# B&R Automation Studio project MotionTestBenchMaster (part 4)

```iecst
(*HRM Type*)

TYPE
	HrmFlr_Type : 	STRUCT
		STS_StatusBits : InStatusBitHrm_Type; (*0*)
		STS_1 : UINT; (*2*)
		STS_2 : UINT; (*4*)
		STS_WDCount : UINT; (*6*)
		CConfig_NR_Heads : UINT; (*8*)
		CConfig_MotorDirection : UINT; (*10*)
		CConfig_GearIn : UDINT; (*12*)
		CConfig_GearOut : UDINT; (*16*)
		CConfig_Res_1 : UINT; (*20*)
		CConfig_Res_2 : UINT; (*22*)
		CConfig_Res_3 : UINT; (*24*)
		CSetup_Mode : UINT; (*26*)
		CSetup_Acc : UINT; (*28*)
		CSetup_Dec : UINT; (*30*)
		CSetup_EDec : UINT; (*32*)
		CSetup_Gearing : UINT; (*34*)
		CSetup_JogSpeed : UINT; (*36*)
		CSetup_JogAcc : UINT; (*38*)
		CSetup_JogDec : UINT; (*40*)
		CSetup_Rpm_at_00K : UINT; (*42*)
		CSetup_Rpm_at_05K : UINT; (*44*)
		CSetup_Rpm_at_10K : UINT; (*46*)
		CSetup_Rpm_at_15K : UINT; (*48*)
		CSetup_Rpm_at_20K : UINT; (*50*)
		CSetup_Rpm_at_25K : UINT; (*52*)
		CSetup_Rpm_at_30K : UINT; (*54*)
		CSetup_Rpm_at_35K : UINT; (*56*)
		CSetup_Rpm_at_40K : UINT; (*58*)
		CSetup_Rpm_at_45K : UINT; (*60*)
		CSetup_Rpm_at_50K : UINT; (*62*)
		CSetup_Rpm_at_55K : UINT; (*64*)
		CSetup_Rpm_at_60K : UINT; (*66*)
		CSetup_Rpm_at_65K : UINT; (*68*)
		CSetup_Rpm_at_70K : UINT; (*70*)
		CSetup_Rpm_at_75K : UINT; (*72*)
		CSetup_Rpm_at_80K : UINT; (*74*)
		CSetup_Rpm_at_85K : UINT; (*76*)
		CSetup_Rpm_at_90K : UINT; (*78*)
		CSetup_Rpm_at_95K : UINT; (*80*)
		CSetup_Rpm_at_100K : UINT; (*82*)
		CSetup_Res_1 : UINT; (*84*)
		CSetup_Res_2 : UINT; (*86*)
		CSetup_Res_3 : UINT; (*88*)
		STS_DiagCode : UINT;
		STS_3 : UINT; (*90*)
		STS_4 : UINT; (*92*)
		STS_ProdSpeedRPM : UINT; (*94*)
		STS_ProdSpeedBPH : UINT; (*96*)
		STS_HeadSpeedRPM : UINT; (*98*)
		STS_5 : UINT; (*100*)
		STS_ActualCurrent : DINT; (*102 v1.7.4*)
		Spare_0 : UINT; (*104*)
		Spare_1 : UINT; (*108*)
		Spare_2 : UINT; (*110*)
		Spare_3 : UINT; (*112*)
		Spare_4 : UINT; (*114*)
		Spare_5 : UINT; (*118*)
		Spare_6 : UINT; (*120*)
		Spare_7 : UINT; (*122*)
		Spare_8 : UINT; (*124*)
		Spare_9 : UINT; (*126*)
	END_STRUCT;
	FlrHrm_Type : 	STRUCT
		CMD_CommandBits : OutCMDHrm_Type; (*0*)
		CMD_1 : UINT; (*2*)
		CMD_2 : UINT; (*4*)
		CMD_3 : UINT; (*6*)
		CConfig_NR_Heads : UINT; (*8*)
		CConfig_MotorDirection : UINT; (*10*)
		CConfig_GearIn : UDINT; (*12*)
		CConfig_GearOut : UDINT; (*16*)
		CConfig_Res_1 : UINT; (*20*)
		CConfig_Res_2 : UINT; (*22*)
		CConfig_Res_3 : UINT; (*24*)
		CSetup_Mode : UINT; (*26*)
		CSetup_Acc : UINT; (*28*)
		CSetup_Dec : UINT; (*30*)
		CSetup_EDec : UINT; (*32*)
		CSetup_Gearing : UINT; (*34*)
		CSetup_JogSpeed : UINT; (*36*)
		CSetup_JogAcc : UINT; (*38*)
		CSetup_JogDec : UINT; (*40*)
		CSetup_Rpm_at_00K : UINT; (*42*)
		CSetup_Rpm_at_05K : UINT; (*44*)
		CSetup_Rpm_at_10K : UINT; (*46*)
		CSetup_Rpm_at_15K : UINT; (*48*)
		CSetup_Rpm_at_20K : UINT; (*50*)
		CSetup_Rpm_at_25K : UINT; (*52*)
		CSetup_Rpm_at_30K : UINT; (*54*)
		CSetup_Rpm_at_35K : UINT; (*56*)
		CSetup_Rpm_at_40K : UINT; (*58*)
		CSetup_Rpm_at_45K : UINT; (*60*)
		CSetup_Rpm_at_50K : UINT; (*62*)
		CSetup_Rpm_at_55K : UINT; (*64*)
		CSetup_Rpm_at_60K : UINT; (*66*)
		CSetup_Rpm_at_65K : UINT; (*68*)
		CSetup_Rpm_at_70K : UINT; (*70*)
		CSetup_Rpm_at_75K : UINT; (*72*)
		CSetup_Rpm_at_80K : UINT; (*74*)
		CSetup_Rpm_at_85K : UINT; (*76*)
		CSetup_Rpm_at_90K : UINT; (*78*)
		CSetup_Rpm_at_95K : UINT; (*80*)
		CSetup_Rpm_at_100K : UINT; (*82*)
		CSetup_Res_1 : UINT; (*84*)
		CSetup_Res_2 : UINT; (*86*)
		CSetup_Res_3 : UINT; (*88*)
		Spare_0 : UINT; (*90*)
		Spare_1 : UINT; (*92*)
		Spare_2 : UINT; (*94*)
		Spare_3 : UINT; (*96*)
		Spare_4 : UINT; (*98*)
		Spare_5 : UINT; (*100*)
		Spare_6 : UINT; (*102*)
		Spare_7 : UINT; (*104*)
		Spare_8 : UINT; (*106*)
		Spare_9 : UINT; (*108*)
		Spare_10 : UINT; (*110*)
		Spare_11 : UINT; (*112*)
		Spare_12 : UINT; (*114*)
		Spare_13 : UINT; (*116*)
		Spare_14 : UINT; (*118*)
		Spare_15 : UINT; (*120*)
		Spare_16 : UINT; (*122*)
		Spare_17 : UINT; (*124*)
		Spare_18 : UINT; (*126*)
	END_STRUCT;
	InStatusBitHrm_Type : 	STRUCT
		ModeAuto : BOOL; (*From AROL HRM Status Bit - Closure Start command request active*)
		Spare0_1 : BOOL; (*From AROL HRM Status Bit -*)
		Enabled : BOOL; (*From AROL HRM Status Bit - Enable command request active*)
		Spare0_3 : BOOL; (*From AROL HRM Status Bit -*)
		GetDiag_DONE : BOOL; (*From AROL HRM Status Bit - System Diagnostic request executed*)
		Spare0_5 : BOOL; (*From AROL HRM Status Bit -*)
		Ready : BOOL; (*From AROL HRM Status Bit - 1: System Active*)
		Alarm : BOOL; (*From AROL HRM Status Bit -PacDrive Controller Alarm*)
		WatchDog : BOOL; (*From AROL HRM Status Bit -WatchDog signal (1s ON and  1s OFF)*)
		HRM_WR : BOOL; (*From AROL HRM Status Bit -HRM is Writing*)
		ConfigNotOK : BOOL; (*From AROL HRM Status Bit -Configuration is not stored in CompactFlash*)
		SetupNotOK : BOOL; (*From AROL HRM Status Bit -Setup is not stored in CompactFlash*)
		Spare1_4 : BOOL; (*From AROL HRM Status Bit -*)
		Spare1_5 : BOOL; (*From AROL HRM Status Bit -*)
		JogForward : BOOL; (*From AROL HRM Status Bit - Manual Command Forward*)
		JogBackward : BOOL; (*From AROL HRM Status Bit - Manual Command Backward*)
	END_STRUCT;
	OutCMDHrm_Type : 	STRUCT
		ClosureStart : BOOL; (*From AROL HRM Status Bit - Closure Start command request active*)
		Spare0_1 : BOOL; (*From AROL HRM Status Bit -*)
		Enable : BOOL; (*From AROL HRM Status Bit - Enable command request active*)
		Spare0_3 : BOOL; (*From AROL HRM Status Bit -*)
		GetDiag : BOOL; (*From AROL HRM Status Bit - System Diagnostic request executed*)
		Spare0_5 : BOOL; (*From AROL HRM Status Bit -*)
		Reset : BOOL; (*From AROL HRM Status Bit - 1: System Active*)
		Spare0_7 : BOOL; (*From AROL HRM Status Bit -PacDrive Controller Alarm*)
		WatchDog : BOOL; (*From AROL HRM Status Bit -WatchDog signal (1s ON and  1s OFF)*)
		StoreConfig : BOOL; (*From AROL HRM Status Bit -HRM is Writing*)
		StoreSetup : BOOL; (*From AROL HRM Status Bit -Configuration is not stored in CompactFlash*)
		Spare1_3 : BOOL; (*From AROL HRM Status Bit -Setup is not stored in CompactFlash*)
		Spare1_4 : BOOL; (*From AROL HRM Status Bit -*)
		Spare1_5 : BOOL; (*From AROL HRM Status Bit -*)
		JogForward : BOOL; (*From AROL HRM Status Bit - Manual Command Forward*)
		JogBackward : BOOL; (*From AROL HRM Status Bit - Manual Command Backward*)
	END_STRUCT;
END_TYPE

(*Syko Multibody Type*)

TYPE
	FlrSikoMbd_Type : 	STRUCT
		SikoCmd : ARRAY[0..5]OF MotorSikoCmd_Type;
		iWatchDog : INT; (*Input WatchDog*)
	END_STRUCT;
	MbdSikoFlr_Type : 	STRUCT
		SikoSts : ARRAY[0..5]OF MotorSikoSts_Type;
		iWatchDog : INT; (*Input WatchDog*)
	END_STRUCT;
	MotorSikoCmd_Type : 	STRUCT
		xEnable : BOOL; (*Enable motor*)
		xReset : BOOL; (*Reset error*)
		xStartPos : BOOL; (*Start positioning*)
		xJogForward : BOOL; (*Jog forward*)
		xJogBackward : BOOL; (*Jog backward*)
		xSetZero : BOOL; (*Set zero position*)
		xWriteParam : BOOL; (*Write parameter*)
		xReadParam : BOOL; (*Read parameter*)
		wCmdSpare : INT; (*Spare commands word*)
		xTargetPosition : DINT; (*Target position*)
		wPositionVelocity : INT; (*Position velocity*)
		wJogVelocity : INT; (*Jog velocity*)
		bCurrentLimit : BYTE; (*Current limit*)
		bSenseOfRotation : BYTE; (*Sense of rotation*)
		wSpare : INT; (*Sense of rotation*)
		wSpare1 : INT; (*Sense of rotation*)
		wSpare2 : INT; (*Sense of rotation*)
		wSpare3 : INT; (*Sense of rotation*)
	END_STRUCT;
	MotorSikoSts_Type : 	STRUCT
		xPowerOk : BOOL; (*Motor power supply is OK*)
		xEnabled : BOOL; (*Motor is enabled*)
		xReady : BOOL; (*Motor is ready*)
		xRunning : BOOL; (*Motor is running*)
		xInPosition : BOOL; (*Motor is in target position*)
		xBatteryWarning : BOOL; (*Motor battery warning error*)
		xError : BOOL; (*Motor generic error*)
		xSpare_1 : BOOL; (*Spare bit*)
		xParamRwBusy : BOOL; (*Parameter read/write operation is busy*)
		xParamRwError : BOOL; (*Parameter read/write operation is in error*)
		xParamRwDone : BOOL; (*Parameter read/write operation is done*)
		wSpareFdbks : UINT; (*Motor actual position*)
		diActualPosition : DINT; (*Motor actual position*)
		wPositionVelocity : INT; (*Jog velocity*)
		wJogVelocity : INT; (*Current limit*)
		bCurrentLimit : BYTE; (*Sense of rotation*)
		bSenseOfRotation : BYTE;
		wSpare0 : INT;
		wSpare1 : INT;
		wSpare2 : {REDUND_UNREPLICABLE} INT;
		wSpare3 : INT;
	END_STRUCT;
	Head_Diagnostic_Type : 	STRUCT
		FaultNumber : USINT;
		StatusOfInverter : USINT;
		TorqueFeedbackOnHead : UINT;
	END_STRUCT;
END_TYPE

(*WATER TREATMENT V4.A.A.1.6.12*)

TYPE
	FlrWtt_Type : 	STRUCT  (*V4.A.A.1.6.12*)
		Alive : BOOL; (*Life bit signal*)
		ProductionRunning : BOOL;
		ProductRequest : BOOL;
		ProductionAlarm : BOOL; (*V4.A.A.1.7.0*)
		BOOL4 : BOOL;
		BOOL5 : BOOL;
		BOOL6 : BOOL;
		BOOL7 : BOOL;
		CipMode : BOOL; (*V4.A.A.1.7.0*)
		CipAlarm : BOOL; (*V4.A.A.1.7.0*)
		CipProductRequest : BOOL; (*V4.A.A.1.7.0*)
		ControlRunning : BOOL; (*V4.A.A.1.7.0*)
	END_STRUCT;
	WttFlr_Type : 	STRUCT  (*V4.A.A.1.6.12*)
		Alive : BOOL; (*Life bit signal*)
		ProductionMode : BOOL;
		ProductAvailable : BOOL;
		FilterCleaning : BOOL;
		OzoneLevelOk : BOOL;
		BOOL5 : BOOL;
		BOOL6 : BOOL;
		BOOL7 : BOOL;
		CipMode : BOOL; (*V4.A.A.1.7.0*)
		CipAlarm : BOOL; (*V4.A.A.1.7.0*)
		CipSending : BOOL; (*V4.A.A.1.7.0*)
		CheckSolutionOk : BOOL; (*V4.A.A.1.7.0*)
	END_STRUCT;
END_TYPE

(*DATA ACQUISITION COMMUNICATION //V4.A.A.1.6.14*)

TYPE
	FlrDaq_Type : 	STRUCT
		Alive : BOOL;
		StopBit : BOOL; (*Common - Stop bit*)
		OperatorPresence : BOOL; (*Common - Operator presence*)
		ModeAuto : BOOL; (*Common - Operator presence*)
		ModeJog : BOOL; (*Common - Operator presence*)
		ModeSetting : BOOL; (*Common - Operator presence*)
		MachineStatus : UINT; (*Common - Machine Status*)
		SKU : UINT; (*Common - SKU*)
		RecipeNumber : UINT; (*Common - Recipe name*)
		Format : UINT; (*Common - Format*)
		Reason : UDINT; (*Common - Reason code that stop the production on machine*)
		ProductionSpeed : UDINT; (*Common - Production speed in CPM (Container per minute)*)
		SetSpeed : UDINT; (*Common - Set speed*)
		InfeedCount : UDINT; (*Filler - Count of infeed container on the machine*)
		ContainersBurstCount : UDINT; (*Filler - Number of Burst container count*)
		LowLevelEjectCount : UDINT;
	END_STRUCT;
	DaqFlr_Type : 	STRUCT
		Alive : BOOL;
	END_STRUCT;
END_TYPE

(*CODER V4.A.A.1.7.0*)

TYPE
	FlrCdr_Type : 	STRUCT  (*V4.A.A.1.7.1*)
		ProductionRunning : BOOL;
		BOOL1 : BOOL;
		BOOL2 : BOOL;
		BOOL3 : BOOL;
		BOOL4 : BOOL;
		BOOL5 : BOOL;
		BOOL6 : BOOL;
		BOOL7 : BOOL;
		BOOL8 : BOOL;
		BOOL9 : BOOL;
	END_STRUCT;
	CdrFlr_Type : 	STRUCT  (*V4.A.A.1.7.1*)
		Alive : BOOL;
		Ready : BOOL; (*Ready*)
		BOOL2 : BOOL;
		BOOL3 : BOOL;
		BOOL4 : BOOL;
		BOOL5 : BOOL;
		BOOL6 : BOOL;
		BOOL7 : BOOL;
		BOOL8 : BOOL;
		BOOL9 : BOOL;
	END_STRUCT;
END_TYPE

(*PST TREATMENT v999hema*)

TYPE
	FlrPst_Type : 	STRUCT
		AliveBit : BOOL; (*Life bit signal*)
		CipSolutionRequest : BOOL;
		CipAlarm : BOOL;
		CipSolutionReturn : BOOL;
		CipRecoveryCompleted : BOOL;
		CipConditionOK : BOOL;
		CipFlipEnded : BOOL;
		CipRunning : BOOL;
		CipDrainCompleted : BOOL;
		CipLevelReached : BOOL;
		RinseRequest : BOOL;
		RinseEnded : BOOL;
		CopRunning : BOOL;
		RinseAfterProdRequest : BOOL;
		RinseAfterProdEnd : BOOL;
		CopHotWaterReq : BOOL;
		CopEnded : BOOL;
		ProductionRunning : BOOL;
		ProductRequest : BOOL;
		ProductionEnded : BOOL;
		ReadyForHeating : BOOL;
		DoserInTemperature : BOOL;
		AVJ201Open : BOOL;
		DoserEmpty : BOOL;
		DoserFull : BOOL;
		ProductRecoveryEnd : BOOL;
		DoserTankLevel : INT;
		DoserTankLevelSP : INT;
		SlurryDoserVolume : INT;
	END_STRUCT;
	PstFlr_Type : 	STRUCT
		AliveBit : BOOL; (*Life bit signal*)
		CipRecipeCompleted : BOOL;
		CipAlarm : BOOL;
		CipProductSending : BOOL;
		CipRecoveryRequest : BOOL;
		CipConditionOK : BOOL;
		CipFlipAllowed : BOOL;
		CipRunning : BOOL;
		CipDrainRequest : BOOL;
		CipRecipeAborted : BOOL;
		CipReturnEnabled : BOOL;
		RinseMode : BOOL;
		RinseSending : BOOL;
		RinseAfterProd : BOOL;
		CopHotWaterSending : BOOL;
		WorkingRinseFromCip : BOOL;
		WorkingHotSanitation : BOOL;
		WorkingCaustic : BOOL;
		WorkingAcid : BOOL;
		WorkingDisinfectant : BOOL;
		ProductionMode : BOOL;
		ProductAvailable : BOOL;
		MinTankLevel : BOOL;
		DrainRequest : BOOL;
		EndProductionReq : BOOL;
		ProductRecoveryRequest : BOOL;
		ProductCompleted : BOOL;
		HeatingWithWater : BOOL;
		ProductAvailableLiters : INT;
		ProductTemperatureSP : INT;
	END_STRUCT;
END_TYPE
```

### MAU_Global.typ
```iecst
(*SafetyCheck*)

TYPE
	SafeLogicStatus_Type : 	STRUCT
		FailSafe : BOOL;
		FirmwareAcknowledge : BOOL;
		NoExecution : BOOL;
		RunDebug : BOOL;
		RunSafe : BOOL;
		SafeKeyExchange : BOOL;
		Scan : BOOL;
		ModuleExchange : UINT;
		ModuleMissing : UINT;
	END_STRUCT;
END_TYPE

(*DUMMY CONTAINERS*)

TYPE
	MAU_DumCon_Type : 	STRUCT
		DataOut : MAU_DumCon_DataOut_Type;
	END_STRUCT;
	MAU_DumCon_DataOut_Type : 	STRUCT
		Idle : BOOL;
		InstallDone : BOOL;
		RemoveDone : BOOL;
		FixSpeedRequest : BOOL;
		MachineStart : BOOL;
		MachineStop : BOOL;
		CounterEnable : BOOL;
		FmcCipMode : BOOL;
		InsControl : BOOL;
		DisControl : BOOL;
		InsertionPistonFault : BOOL;
		DmcInsCsrPositioning : BOOL;
		DmcDisCsrPositioning : BOOL;
		LftCenteringCupUp : BOOL;
		LftCenteringCupDownOnCip : BOOL;
		ContainerStop : BOOL; (*//1.63*)
		DmcManualModeActive : BOOL; (*v1.6*)
		FlrToCipHeight : BOOL; (*v999*)
		Sector1DownToCip : BOOL; (*v999*)
		Sector2DownToCip : BOOL; (*v999*)
		Sector1DownToProd : BOOL; (*v999*)
		Sector2DownToProd : BOOL; (*v999*)
		Sector1OnlyRotToCip : BOOL;
		Sector2OnlyRotToCip : BOOL;
		Sector2OnlyRotToProd : BOOL;
		Sector1OnlyRotToProd : BOOL;
		DmcUpInProgress : BOOL;
		FillerReversePosReq : BOOL; (*v999*)
		FillerFirstHalfPosReq : BOOL; (*v999*)
		FirstHalfDisDmcControl : BOOL; (*v999*)
		FillerSecondHalfInserted : BOOL;
		FillerFirstHalfRemoved : BOOL;
		FillerFirstHalfInserted : BOOL;
		FillerSecondHalfRemoved : BOOL;
		SecondHalfDisDmcControl : BOOL; (*v999*)
		FirstHalfInsDmcControl : BOOL; (*V999*)
		ManualAirDischarge : BOOL; (*v999*)
		FmcPhasingReq : BOOL; (*v999*)
		FmcInOperational : BOOL; (*v999*)
		FirstHalfInstControl : BOOL; (*v999*)
		SecondHalfInsDmcControl : BOOL; (*v999*)
		FillerSecondHalfPosReq : BOOL; (*v999*)
		FillerSecondReversePosReq : BOOL; (*v999*)
		SectorDiscargePressure : BOOL; (*v999*)
		ContainerLiftAirDischarge : BOOL;
		ManualModeEnableSec2 : BOOL;
		ManualModeEnableSec1 : BOOL;
		DmcManualOperationEn : BOOL; (*V4.A.A.1.7.1*)
		Dba_Sector2ManDownReq : BOOL;
		Dba_Sector1ManDownReq : BOOL;
		ManModeDisControlSec1 : BOOL;
		CycleFmcInError : BOOL;
		CycleAborted : BOOL;
		ReducePressureToUp : BOOL;
		TankCammaToProdHeight : BOOL;
		ManModeDisControlSec2 : BOOL;
	END_STRUCT;
END_TYPE

(*LIFT CONTAINERS*)

TYPE
	MAU_LftCon_Type : 	STRUCT
		DataOut : MAU_LftCon_DataOut_Type;
	END_STRUCT;
	MAU_LftCon_DataOut_Type : 	STRUCT
		LiftContainerUp : BOOL := TRUE;
		CenteringCupUp : BOOL;
		CenteringCupDownOnCip : BOOL;
		CenteringCupAirOn : BOOL := TRUE;
		CenteringCupUpTime : UINT;
		WaterReq : BOOL;
	END_STRUCT;
END_TYPE

(*TRAY*)

TYPE
	MAU_Tray_Type : 	STRUCT  (*v1.4*)
		DataOut : MAU_Tray_DataOut_Type;
	END_STRUCT;
	MAU_Tray_DataOut_Type : 	STRUCT  (*v1.4*)
		ContainerStop : BOOL; (*//1.63*)
		TrayInPosition : BOOL;
	END_STRUCT;
END_TYPE

(*UPS*)

TYPE
	MAU_Ups_Type : 	STRUCT
		DataOut : MAU_Ups_DataOut_Type;
	END_STRUCT;
	MAU_Ups_DataOut_Type : 	STRUCT
		PowerOffTime : UINT;
	END_STRUCT;
END_TYPE

(*AUX  V1.7.2*)

TYPE
	MAU_Aux_Type : 	STRUCT
		DataOut : MAU_Aux_DataOut_Type;
	END_STRUCT;
	MAU_Aux_DataOut_Type : 	STRUCT
		ContainerStop : BOOL;
		EjectionRequest : BOOL;
	END_STRUCT;
END_TYPE

(*SCHEDULER //v1.7.4*)

TYPE
	MAU_Scheduler_Type : 	STRUCT
		DataOut : MAU_Scheduler_DataOut_Type;
	END_STRUCT;
	MAU_Scheduler_DataOut_Type : 	STRUCT
		AlarmMSInternal : UINT;
		AlarmCSRInternal : UINT;
		AlarmCSAInternal : UINT;
		AlarmMSExternal : UINT;
		AlarmCSRExternal : UINT;
		AlarmCSRExternalDw : UINT;
		AlarmCSAExternal : UINT;
		AlarmCSAExternalDw : UINT;
		AlarmInternalOMAC : UINT; (*V1.7.4*)
		AlarmExternalOMAC : UINT; (*V1.7.4*)
	END_STRUCT;
END_TYPE
```

### MC_Global.typ
```iecst
(*Motion Interface Data Type*)

TYPE
	ST_MotionInterface : 	STRUCT
		Safety : ST_SafetyInterface;
		Network : ST_NetworkInterface;
	END_STRUCT;
END_TYPE

(*Interfaces*)

TYPE
	ST_SafetyInterface : 	STRUCT  (*Process-Motion safety interface*)
		Filler : ST_FillerSafetyInterface; (*Filler input/output safety interface*)
		Inlet : ST_InletSafetyInterface; (*Inlet input/output safety interface*)
		Outlet : ST_OutletSafetyInterface; (*Outlet input/output safety interface*)
	END_STRUCT;
	ST_NetworkInterface : 	STRUCT  (*Process-Motion network interface*)
		Machine : ST_MachineInterface; (*Machine input output interface*)
		Inlet : ST_InletInterface; (*Inlet input/output interface*)
		Filler : ST_FillerInterface; (*Filler input/output interface*)
		Outlet : ST_OutletInterface; (*Outlet input/output interface*)
	END_STRUCT;
END_TYPE

(*Machine*)

TYPE
	ST_MachineInterface : 	STRUCT  (*Machine input/output interface structure*)
		Commands : ST_MachineCommandsInterface; (*Machine commands structure*)
		Parameters : ST_MachineParametersInterface; (*Machine parameter structure*)
		Status : ST_MachineStatusInterface; (*Machine status structure*)
		Exceptions : ST_MachineExceptionsInterface; (*Machine exception structure*)
	END_STRUCT;
	ST_MachineCommandsInterface : 	STRUCT  (*Machine commands*)
		HandShakeIn : BOOL; (*Not Used on Full B&R Machines.*)
		MachineStart : BOOL; (*Start commands. When this signal falls the machine start a deceleration ramp.*)
		AlarmReset : BOOL; (*Reset motion alarm command.*)
		MachineQuickStop : BOOL; (*Machine quick stop. This signal has to be set to 1 during normal operation. If this signal will fall a quick stop is performed.*)
		SynchroDisengage : BOOL; (*The interfaces between filler machine and other machines. This value is taken in account only if the CFG_MC.Generic.DisengageImmediately is set.*)
		JogPushButton : BOOL; (*Jog Push Button.*)
		DisableRinserAxis : BOOL; (*The selected axis is disabled rotation V4.A.A.1.7.0*)
		DisableSelectedAxis : BOOL; (*The selected axis is disabled. This operation works only in emergency.*)
		BrakeReleaseModalityRequest : BOOL; (*Brake Release modality request on selected axis.*)
		SelectiveHomeModalityRequest : BOOL; (*Home modality request on selected axis / external reference.*)
		AllAxesHomeModalityRequest : BOOL; (*Homing of all axes - Not Implemented yet.*)
		MultiModalityRequest : BOOL; (*Multi modality selected in order to send the command directly to the module.*)
		PositioningModalityRequest : BOOL; (*Positioning Modality Request.*)
		AutoModalityRequest : BOOL; (*Auto (stand alone) Modality Request.*)
		AutoCombiModalityRequest : BOOL; (*Combi modality request. The machine will follow an external reference.*)
		JogMachineModalityRequest : BOOL; (*Jog modality request.*)
		StepByStepSingleAxisRevModReq : BOOL; (*Single Axis Step By Step Reverse modality request V999*)
		StepByStepSingleAxisModReq : BOOL; (*Single Axis Step By Step modality request V4.A.A.1.7.0*)
		StepByStepModalityRequest : BOOL; (*Step By Step modality request.*)
		EndlessModalityRequest : BOOL; (*Endless modality request - not implemented yet.*)
		ThirdPartMotStatSetupModReq : BOOL; (*Third Party Motor Static Modality Request - not implemented yet.*)
		ThirdPartMotDynSetupModReq : BOOL; (*Endless modality request- not implemented yet.*)
		InMotionTimerModReq : BOOL; (*InMotion Timer function request on active axis.*)
		VelocityModalityRequest : BOOL; (*Velocity Modality Request on actis axis.*)
		OkToDisengage : BOOL; (*The interface is free.*)
		CombiSynchroStop : BOOL; (*Combi Synchro Stop. The machine will continue to turn at constant speed.*)
		MasterEncoderPositionValid : BOOL; (*The position of the master encoder is valid. In case of FALSE in combi mode a Quick Stop is performed.*)
		OnePitchShiftCommand : BOOL; (*One Pitch Shift in combi mode for the "One container every two steps" option.*)
		KochModuleReady : BOOL; (*Where present this variable is linked to the Koch module status*)
		FanSeamerFeedback : BOOL;
		FanSeamerOn : BOOL;
		FanSeamerThermalOverload : BOOL;
	END_STRUCT;
	ST_MachineStatusInterface : 	STRUCT  (*Machine status*)
		HandshakeOut : BOOL; (*Not Used on Full B&R Machines.*)
		MachineHomed : BOOL; (*All axis on the machine are homed.*)
		MachineInPosition : BOOL; (*All axis on the machine are in position.*)
		MachineRunning : BOOL; (*At least one axis is running.*)
		MachineSynchro : BOOL; (*The machine is internally synchronized.*)
		MachineStartFbk : BOOL; (*Feedback of the machine start. See timechart for details.*)
		AutoCmdFeedback : BOOL; (*Auto Modality feedback (?)*)
		JogCmdFeedback : BOOL; (*Jog Modality feedback (?)*)
		AxisNoOp : BOOL;
		MachineIE : BOOL; (*Machine Powered.*)
		MachinePowered : BOOL; (*Machine Powered.*)
		ModuleNotInitialized : BOOL; (*Master Module Not Initialized; the master module isn't initialized. PowerOn the module. 1.7.2a*)
		EnableStart : BOOL; (*Enable start . All motion conditions are ready for the rotation.*)
		EnableAuto : BOOL; (*Enable Auto . All motion conditions are verifier in order to enable auto modality.*)
		EnableEndless : BOOL; (*Enable Endless . All condition are verified in order to have the endless modality.*)
		EnableBrakeRelease : BOOL; (*Enable Brake Release . All condition are verified in order to release the brake.*)
		EnablePositioning : BOOL; (*Enable Positioning . All condition are verified in order to make a positioning.*)
		EnableHoming : BOOL; (*Enable Homing . All condition are verified in order to make the homing of an axis.*)
		EnableCombi : BOOL; (*Enable Combi . All condition are verified in order to enable the combi modality.*)
		EnableMulti : BOOL; (*Enable Multi . All condition are verified in order to enable the spliltted modalities.*)
		EnableSlowMotion : BOOL; (*Enable Slow Motion. All condition are verified in order to enable the slow motion.*)
		EnableStepByStep : BOOL; (*Enable StepByStep . All condition are verified in order to enable the step by step modality.*)
		EnableJog : BOOL; (*Enable Jog . All condition are verified in order to enable the jog modality.*)
		EnableInMotionTimer : BOOL; (*Enable InMotion Timer . All condition are verified in order to enable the in motion timer.*)
		EnableAxisEnable : BOOL; (*Enable AxisEnable Button . All condition are verified in order to enable or disable the axis.*)
		EnableVelocity : BOOL; (*Enable Velocity . All condition are verified in order to make a velociy.*)
		ThirdPartMotStatSetupButton : BOOL; (*Enable thirdy party motor setup. All condition are verified in order to enable the third party static motor setup.*)
		ThirdPartMotDynSetupButton : BOOL; (*Enable thirdy party motor setup. All condition are verified in order to enable the third party dinamic motor setup.*)
		InductionMotSetupButton : BOOL; (*Induction motor setup. All condition are verified in order to enable the third party dinamic motor setup.*)
		NoModalityActive : BOOL; (*No modality selected on motion control.*)
		SelectiveHomeModalityActive : BOOL; (*Selective home modality active.*)
		VelocityModalityActive : BOOL; (*Velocity modality active on axis with velocity control.*)
		PositioningModalityActive : BOOL; (*Positioning modality active.*)
		JogModalityActive : BOOL; (*Jog modality active.*)
		BrakeReleaseModalityActive : BOOL; (*Brake release modality active.*)
		StepByStepSingleAxisRevModActive : BOOL; (*Single Axis Step by step Reverse modality active. V999*)
		StepByStepSingleAxisModeActive : BOOL; (*Single Axis Step by step modality active. V4.A.A.1.7.0*)
		StepByStepModalityActive : BOOL; (*Step by step modality active.*)
		EndlessModalityActive : BOOL; (*Endless modality active.*)
		MultiModalityActive : BOOL; (*Multi modality active. All modules are working indipendently.*)
		ThirdPartMotStatSetupModAct : BOOL; (*Third party motor static setup active.*)
		ThirdPartMotDynSetupModAct : BOOL; (*Third party motor dynamic setup active.*)
		InductionMotSetupActive : BOOL; (*Induction motor setup active.*)
		AutoModalityActive : BOOL; (*Auto modality active.*)
		AutoCombiModalityActive : BOOL; (*Auto combi modality active.*)
		CombiSynchroStopDone : BOOL; (*Combi synchro stop done.*)
		CombiSynchronized : BOOL; (*Combi synchron. All axis are syncrhonized with the external reference.*)
		CombiSynchroInProgress : BOOL; (*Combi synchro in progress.*)
		CombiFixedSpeed : BOOL; (*Combi fixed speed. The combi after a request is running in continous motion.*)
		InMotionTimerDone : BOOL; (*The in motion timer movement has beed done.*)
		OnePitchShiftDone : BOOL;
		MachineClockA : BOOL; (*Main machine clock.*)
		MachineClockB : BOOL; (*Main machine clock.*)
		Clock01 : BOOL; (*Clock 1 at disposal.*)
		Clock02 : BOOL; (*Clock 2 at disposal.*)
		Clock03 : BOOL; (*Clock 3 at disposal.*)
		Clock04 : BOOL; (*Clock 4 at disposal.*)
		Clock05 : BOOL; (*Clock 5 at disposal.*)
		Clock06 : BOOL; (*Clock 6 at disposal.*)
		Clock07 : BOOL; (*Clock 7 at disposal.*)
		Clock08 : BOOL; (*Clock 8 at disposal.*)
		Clock09 : BOOL; (*Clock 9 at disposal.*)
		Clock10 : BOOL; (*Clock 10 at disposal.*)
		Clock11 : BOOL; (*Clock 11 at disposal. v999hema*)
		Clock01AdvStep : BOOL; (*Clock 2 at disposal.*)
		Clock02AdvStep : BOOL; (*Clock 2 at disposal.*)
		Clock03AdvStep : BOOL; (*Clock 3 at disposal.*)
		Clock04AdvStep : BOOL; (*Clock 4 at disposal.*)
		Clock05AdvStep : BOOL; (*Clock 5 at disposal.*)
		Clock06AdvStep : BOOL; (*Clock 6 at disposal.*)
		Clock07AdvStep : BOOL; (*Clock 7 at disposal.*)
		Clock08AdvStep : BOOL; (*Clock 8 at disposal.*)
		Clock09AdvStep : BOOL; (*Clock 9 at disposal.*)
		Clock10AdvStep : BOOL; (*Clock 10 at disposal.*)
		Clock11AdvStep : BOOL; (*Clock 11 at disposal. v999hema*)
		AxisSelectedForEndless : INT; (*Axis selected for endlessfeed feedback.*)
		SpeedForAxisSelectedEndless : INT; (*Speed selected for endlessfeed feedback.*)
		ActualSpeed : REAL; (*Machine velocity [bph].*)
		MachineMaxSpeed : REAL; (*Machine Max velocity [bph].*)
		MachinePitch : REAL; (*Machine Pitch [teens of mm].*)
	END_STRUCT;
	ST_MachineParametersInterface : 	STRUCT  (*Machine parameters*)
		AxisSelectedOnHmi : INT; (*Axis Selected On Hmi*)
		StepNumber : INT; (*Number of step for StepByStep movement [n]*)
		ManualVelocity : UINT;
		JogSpeed : REAL; (*Jog velocity [cph]*)
		AutoSpeed : REAL; (*Auto Velocity [cph]*)
		AutoAccelerationTime : REAL; (*Deceleration Time [s]*)
		AutoDecelerationTime : REAL; (*Acceleration Time [s]*)
		OffsetPositioning : REAL; (*Positioning Offset [mm]*)
		OffsetHoming : REAL; (*Homing Offset - not implemented yet*)
		StopPosition : REAL; (*Stop Position [mm]*)
		InMotionTimerValue : REAL; (*In motion timer value [mm]*)
		Cam01OnValue : REAL; (*Cam01 On Value*)
		Cam01OffValue : REAL; (*Cam01 Off Value*)
		Cam01AdvTime : REAL; (*Cam01 Advance Time*)
		Cam01Pulse : USINT; (*Cam01 Pulse number*)
		Cam02OnValue : REAL; (*Cam02 On Value*)
		Cam02OffValue : REAL; (*Cam02 Off Value*)
		Cam02AdvTime : REAL; (*Cam02 Advance Time*)
		Cam02Pulse : USINT; (*Cam02 Pulse number*)
		Cam03OnValue : REAL; (*Cam03 On Value*)
		Cam03OffValue : REAL; (*Cam03 Off Value*)
		Cam03AdvTime : REAL; (*Cam03 Advance Time*)
		Cam03Pulse : USINT; (*Cam03 Pulse number*)
		Cam04OnValue : REAL; (*Cam04 On Value*)
		Cam04OffValue : REAL; (*Cam04 Off Value*)
		Cam04AdvTime : REAL; (*Cam04 Advance Time*)
		Cam04Pulse : USINT; (*Cam04 Pulse number*)
		Cam05OnValue : REAL; (*Cam05 On Value*)
		Cam05OffValue : REAL; (*Cam05 Off Value*)
		Cam05AdvTime : REAL; (*Cam05 Advance Time*)
		Cam05Pulse : USINT; (*Cam05 Pulse number*)
		Cam06OnValue : REAL; (*Cam06 On Value*)
		Cam06OffValue : REAL; (*Cam06 Off Value*)
		Cam06AdvTime : REAL; (*Cam06 Advance Time*)
		Cam06Pulse : USINT; (*Cam06 Pulse number*)
		Cam07OnValue : REAL; (*Cam07 On Value*)
		Cam07OffValue : REAL; (*Cam07 Off Value*)
		Cam07AdvTime : REAL; (*Cam07 Advance Time*)
		Cam07Pulse : USINT; (*Cam07 Pulse number*)
		Cam08OnValue : REAL; (*Cam08 On Value*)
		Cam08OffValue : REAL; (*Cam08 Off Value*)
		Cam08AdvTime : REAL; (*Cam08 Advance Time*)
		Cam08Pulse : USINT; (*Cam08 Pulse number*)
		Cam09OnValue : REAL; (*Cam09 On Value*)
		Cam09OffValue : REAL; (*Cam09 Off Value*)
		Cam09AdvTime : REAL; (*Cam09 Advance Time*)
		Cam09Pulse : USINT; (*Cam09 Pulse number*)
		Cam10OnValue : REAL; (*Cam10 On Value*)
		Cam10OffValue : REAL; (*Cam10 Off Value*)
		Cam10AdvTime : REAL; (*Cam10 Advance Time*)
		Cam10Pulse : USINT; (*Cam10 Pulse number*)
		Cam11OffValue : REAL; (*Cam11 Off Value v999hema*)
		Cam11AdvTime : REAL; (*Cam11 Advance Time*)
		Cam11OnValue : REAL; (*Cam11 On Value*)
		Cam11Pulse : USINT; (*Cam11 Pulse number*)
		AxisSelectedForEndless : INT; (*Axis Selected for EndlessFeed - not implemented yet*)
		SpeedForAxisSelectedEndless : INT; (*Speed For Axis Selected for EndlessFeed - not implemented yet*)
		MachinePitch : REAL; (*Machine Pitch [teens of mm]*)
	END_STRUCT;
	ST_MachineExceptionsInterface : 	STRUCT  (*Machine exceptions*)
		Fault : BOOL; (*Generic motion exception.*)
		TrackErrorDataException : BOOL;
		HmiChecksumException : BOOL; (*Hmi parameter checksum exception. Used in standalone applications.*)
		PowerSupplyLowMachineException : BOOL; (*Power supply voltage too low exception.*)
		DcBusLowMachineException : BOOL; (*DcBus too low exception.*)
		PhaseMonitoringException : BOOL; (*Phase monitoring exception*)
		KochModuleNotReady : BOOL; (*Where is installed the Koch module ins't correctly charged.*)
		FanSeamearFault : BOOL;
		ExcessiveVelocityException : BOOL; (*Excessive velocity exception (not implemented yet).*)
		ExcessiveAccException : BOOL; (*Excessive acceleration exception (not implemented yet).*)
		NoAxisEnabledException : BOOL; (*No axis enable exception (not implemented yet).*)
		HomingException : BOOL; (*Machine not homed exception.*)
		BleederException : BOOL; (*Bleeder exception. A bleeder error has occurred.*)
		NegativeSpeedBlowerException : BOOL; (*The reference has a negative speed.*)
		CombiException : BOOL;
		InitEncoderException : BOOL;
		FaultCamGeneration : BOOL; (*V1.7.2*)
		StopBlowerException : BOOL;
	END_STRUCT;
END_TYPE

(*Inlet module*)

TYPE
	ST_InletInterface : 	STRUCT  (*Inlet module input/output interface structure*)
		Commands : ST_InletCommands; (*Inlet commands structure*)
		Parameters : ST_InletParameters; (*Inlet parameters structure*)
		Status : ST_InletStatus; (*Inlet status structure*)
		Exceptions : ST_InletExceptions; (*Inlet exception structure*)
	END_STRUCT;
	ST_InletCommands : 	STRUCT  (*Inlet module commands*)
		AutoInletModule : BOOL; (*Auto modality request for auto module in multi mode.*)
		JogInletModule : BOOL; (*Jog modality request for auto module in multi mode.*)
		QuickStopInletModule : BOOL; (*Quick stop on Inlet module; quick stop not active signal 1.*)
		StartInletModule : BOOL; (*Start on Inlet module.*)
		JogPushButtonInletModule : BOOL; (*Jog push button for Inlet module.*)
		SlowMotionBackward : BOOL; (*Slow motion backward on Inlet module.*)
		SlowMotionForward : BOOL; (*Slow motion forward on Inlet module.*)
		AbsolutePositionSensor : BOOL;
		VelocityAxisStop : BOOL;
	END_STRUCT;
	ST_InletStatus : 	STRUCT  (*Inlet module parameters*)
		ModuleHomed : BOOL; (*Inlet Module Homed; all axes are homed.*)
		ModuleInPosition : BOOL; (*Inlet Module In Position; all axes are standstill and in position.*)
		ModuleRunning : BOOL; (*Inlet Module Running; at least one axis is not standstill.*)
		ModulePowered : BOOL; (*Inlet Module Powered; Inlet module is enabled from a safety point of view.*)
		EnableAutoModality : BOOL; (*Inlet Module Enable Auto Modality; during machine multi mode all condition are valid for enabling the Auto modality.*)
		EnableJogModality : BOOL; (*Inlet Module Enable Auto Modality; during machine multi mode all condition are valid for enabling the Jog modality.*)
		ModuleJogActive : BOOL; (*Inlet Module Jog Active; the jog modality on the Inlet module is active.*)
		AutoActive : BOOL; (*Inlet Module Auto Active; the auto modality on the Inlet module is active.*)
		SlowMotionActive : BOOL; (*Inlet Module Slow Motion Active; the slow motion on the Inlet module is active.*)
		JogCmdFeedback : BOOL; (*Inlet Module Jog Command Feedback.*)
		AutoCmdFeedback : BOOL; (*Inlet Module Auto Command Feedback.*)
		ModuleNotInitialized : BOOL; (*Inlet Module Not Initialized; the Inlet module isn't initialized. PowerOn the module.*)
		ModuleReal : BOOL; (*Inlet Module Real; at least one axis is real on the Inlet module.*)
		In01Real : BOOL; (*Axis Inlet01 on filler module is real.*)
		In02Real : BOOL; (*Axis Inlet02 on filler module is real.*)
		In03Real : BOOL; (*Axis Inlet03 on filler module is real.*)
		In04Real : BOOL; (*Axis Inlet04 on filler module is real.*)
		In05Real : BOOL; (*Axis Inlet05 on filler module is real.*)
		In06Real : BOOL; (*Axis Inlet06 on filler module is real.*)
		MainAxisReal : BOOL; (*Main axis on filler module is real.*)
		Velocity : REAL; (*Auto speed for Inlet module [bph].*)
		AbsolutePosition : LREAL;
		AbsolutePositionValid : BOOL;
	END_STRUCT;
	ST_InletParameters : 	STRUCT  (*Inlet module exception*)
		AutoSpeedInletModule : REAL; (*Auto speed for inlet module [bph]*)
		AbsolutePositionValveOffset : UINT;
		ConveyorKs : REAL;
		WheelValvesNumber : UINT;
		TorqueError : CFG_InletTorque_Type;
	END_STRUCT;
	ST_InletExceptions : 	STRUCT  (*Inlet module exception*)
		MainAxisTrackException : BOOL; (*Main Axis Inlet module track error exception.*)
		MainAxisHomeException : BOOL; (*Main Axis Inlet module home exception.*)
		MainAxisTorqueException : BOOL; (*Main Axis Inlet module torque exception.*)
		MainAxisDriveException : BOOL; (*Main Axis Inlet module drive exception.*)
		MainAxisTemperatureError : BOOL; (*Main Axis Inlet module temperature exception.*)
		MainAxisSafetyException : BOOL; (*Main Axis Inlet module safety exception.*)
		MainAxisNotInOpException : BOOL; (*Main Axis Inlet module not in operational exception.*)
		Inlet01TrackException : BOOL; (*Inlet01 track error exception.*)
		Inlet01HomeException : BOOL; (*Inlet01 home exception.*)
		Inlet01TorqueException : BOOL; (*Inlet01 torque exception.*)
		Inlet01DriveException : BOOL; (*Inlet01 drive exception.*)
		Inlet01TemperatureError : BOOL; (*Inlet01 temperature exception.*)
		Inlet01SafetyException : BOOL; (*Inlet01 safety exception.*)
		Inlet01NotInOpException : BOOL; (*Inlet01 not in operational exception.*)
		Inlet02TrackException : BOOL; (*Inlet02 track error exception.*)
		Inlet02HomeException : BOOL; (*Inlet02 home exception.*)
		Inlet02TorqueException : BOOL; (*Inlet02 torque exception.*)
		Inlet02DriveException : BOOL; (*Inlet02 drive exception.*)
		Inlet02TemperatureError : BOOL; (*Inlet02 temperature exception.*)
		Inlet02SafetyException : BOOL; (*Inlet02 safety exception.*)
		Inlet02NotInOpException : BOOL; (*Inlet02 not in operational exception.*)
		Inlet03TrackException : BOOL; (*Inlet03 track error exception.*)
		Inlet03HomeException : BOOL; (*Inlet03 home exception.*)
		Inlet03TorqueException : BOOL; (*Inlet03 torque exception.*)
		Inlet03DriveException : BOOL; (*Inlet03 drive exception.*)
		Inlet03TemperatureError : BOOL; (*Inlet03 temperature exception.*)
		Inlet03SafetyException : BOOL; (*Inlet03 safety exception.*)
		Inlet03NotInOpException : BOOL; (*Inlet03 not in operational exception.*)
		Inlet04TrackException : BOOL; (*Inlet04 track error exception.*)
		Inlet04HomeException : BOOL; (*Inlet04 home exception.*)
		Inlet04TorqueException : BOOL; (*Inlet04 torque exception.*)
		Inlet04DriveException : BOOL; (*Inlet04 drive exception.*)
		Inlet04TemperatureError : BOOL; (*Inlet04 temperature exception.*)
		Inlet04SafetyException : BOOL; (*Inlet04 safety exception.*)
		Inlet04NotInOpException : BOOL; (*Inlet04 not in operational exception.*)
		Inlet05TrackException : BOOL; (*Inlet05 track error exception.*)
		Inlet05HomeException : BOOL; (*Inlet05 home exception.*)
		Inlet05TorqueException : BOOL; (*Inlet05 torque exception.*)
		Inlet05DriveException : BOOL; (*Inlet05 drive exception.*)
		Inlet05TemperatureError : BOOL; (*Inlet05 temperature exception.*)
		Inlet05SafetyException : BOOL; (*Inlet05 safety exception.*)
		Inlet05NotInOpException : BOOL; (*Inlet05 not in operational exception.*)
		Inlet06TrackException : BOOL; (*Inlet06 track error exception.*)
		Inlet06HomeException : BOOL; (*Inlet06 home exception.*)
		Inlet06TorqueException : BOOL; (*Inlet06 torque exception.*)
		Inlet06DriveException : BOOL; (*Inlet06 drive exception.*)
		Inlet06TemperatureError : BOOL; (*Inlet06 temperature exception.*)
		Inlet06SafetyException : BOOL; (*Inlet06 safety exception.*)
		Inlet06NotInOpException : BOOL; (*Inlet06 not in operational exception.*)
	END_STRUCT;
END_TYPE

(*Filler module*)

TYPE
	ST_FillerInterface : 	STRUCT  (*Filler module input/output interface structure*)
		Commands : ST_FillerCommands; (*Filler commands structure*)
		Parameters : ST_FillerParameters; (*Filler parameters structure*)
		Status : ST_FillerStatus; (*Filler status structure*)
		Exceptions : ST_FillerExceptions; (*Filler exceptions structure*)
	END_STRUCT;
	ST_FillerCommands : 	STRUCT  (*Filler module commands structure*)
		AutoFillerModule : BOOL; (*Auto modality request for auto module in multi mode.*)
		JogFillerModule : BOOL; (*Jog modality request for auto module in multi mode.*)
		QuickStopFillerModule : BOOL; (*Quick stop on filler module; quick stop not active signal 1.*)
		StartFillerModule : BOOL; (*Start on filler module.*)
		JogPushButtonFillerModule : BOOL; (*Jog push button for filler module.*)
		FillerAbsolutePositionSensor : BOOL;
		MotorDisableIndex : ARRAY[CST_FirstFillerModuleAxis..CST_LastFillerModuleAxis]OF BOOL; (*v999 test*)
		DisableFillerAxis : BOOL; (*v999hema*)
		DisableDoserAxis : BOOL; (*V4.A.A.1.7.0*)
		DisableRinserAxis : BOOL; (*V4.A.A.1.7.0*)
		RinserAbsolutePositionSensor : BOOL;
		CapperAbsolutePositionSensor : BOOL;
		CrownerAbsolutePositionSensor : BOOL;
		DoserAbsolutePositionSensor : BOOL;
		VelocityAxisStop : BOOL;
		StepByStepModalityRequest : BOOL;
	END_STRUCT;
	ST_FillerStatus : 	STRUCT  (*Filler module status structure*)
		ModuleHomed : BOOL; (*Filler Module Homed; all axes are homed.*)
		ModuleInPosition : BOOL; (*Filler Module In Position; all axes are standstill and in position.*)
		ModuleRunning : BOOL; (*Filler Module Running; at least one axis is not standstill.*)
		ModulePowered : BOOL; (*Filler Module Powered; filler module is enabled from a safety point of view.*)
		EnableAutoModality : BOOL; (*Filler Module Enable Auto Modality; during machine multi mode all condition are valid for enabling the Auto modality.*)
		EnableJogModality : BOOL; (*Filler Module Enable Auto Modality; during machine multi mode all condition are valid for enabling the Jog modality.*)
		StepByStepModalityActive : BOOL;
		ModuleJogActive : BOOL; (*Filler Module Jog Active; the jog modality on the filler module is active.*)
		AutoActive : BOOL; (*Filler Module Auto Active; the auto modality on the filler module is active.*)
		SlowMotionActive : BOOL; (*Filler Module Slow Motion Active; the slow motion on the filler module is active.*)
		JogCmdFeedback : BOOL; (*Filler Module Jog Command Feedback.*)
		AutoCmdFeedback : BOOL; (*Filler Module Auto Command Feedback.*)
		ModuleNotInitialized : BOOL; (*Filler Module Not Initialized; the filler module isn't initialized. PowerOn the module.*)
		ModuleReal : BOOL; (*Filler Module Real; at least one axis is real on the filler module.*)
		FillerAbsolutePositionValid : BOOL;
		RinserAbsolutePositionValid : BOOL;
		CapperAbsolutePositionValid : BOOL;
		CrownerAbsolutePositionValid : BOOL;
		DoserAbsolutePositionValid : BOOL;
		AxisDisabledFeedBack : ARRAY[CST_FirstFillerModuleAxis..CST_LastFillerModuleAxis]OF BOOL; (*v999 test*)
		DoserAxisDisabled : BOOL; (*v999hema*)
		FillerAxisDisabled : BOOL; (*v999hema*)
		RinserAxisDisabled : BOOL; (*Rinser axis disable answer V4.A.A.1.7.0*)
		In01Real : BOOL; (*Axis Inlet01 on filler module is real.*)
		In02Real : BOOL; (*Axis Inlet02 on filler module is real.*)
		In03Real : BOOL; (*Axis Inlet03 on filler module is real.*)
		In04Real : BOOL; (*Axis Inlet04 on filler module is real.*)
		In05Real : BOOL; (*Axis Inlet05 on filler module is real.*)
		In06Real : BOOL; (*Axis Inlet06 on filler module is real.*)
		In07Real : BOOL; (*Axis Inlet07 on filler module is real.*)
		In08Real : BOOL; (*Axis Inlet08 on filler module is real.*)
		In09Real : BOOL; (*Axis Inlet09 on filler module is real.*)
		In10Real : BOOL; (*Axis Inlet10 on filler module is real.*)
		CarouselReal : BOOL; (*Axis Carousel on filler module is real.*)
		Out01Real : BOOL; (*Axis Outlet01 on filler module is real.*)
		Out02Real : BOOL; (*Axis Outlet02 on filler module is real.*)
		Out03Real : BOOL; (*Axis Outlet03 on filler module is real.*)
		Out04Real : BOOL; (*Axis Outlet04 on filler module is real.*)
		Out05Real : BOOL; (*Axis Outlet05 on filler module is real.*)
		Out06Real : BOOL; (*Axis Outlet06 on filler module is real.*)
		Velocity : REAL; (*Filler module actual velocity [bph]*)
		FillerAbsolutePosition : LREAL;
		RinserAbsolutePosition : LREAL;
		CapperAbsolutePosition : LREAL;
		CrownerAbsolutePosition : LREAL;
		DoserAbsolutePosition : LREAL;
	END_STRUCT;
	ST_FillerParameters : 	STRUCT  (*Filler module parameters structure*)
		AutoSpeedFillerModule : REAL; (*Auto speed for filler module [bph]*)
		FillerStepsNumber : UINT;
		RinserStepsNumber : UINT;
		CapperStepsNumber : UINT;
		CrownerStepsNumber : UINT;
		DoserStepsNumber : UINT;
		FillerAbsolutePositionOffset : UINT;
		RinserAbsolutePositionOffset : UINT;
		CapperAbsolutePositionOffset : UINT;
		CrownerAbsolutePositionOffset : UINT;
		DoserAbsolutePositionOffset : UINT;
		InletConveyorKs : REAL;
		OutletConveyorKs : REAL;
		StepNumber : INT; (*Number of step for StepByStep movement [n]*)
		TorqueError : CFG_FillerTorque_Type;
	END_STRUCT;
	ST_FillerExceptions : 	STRUCT  (*Filler module exception structure*)
		Inlet01TrackException : BOOL; (*Inlet01 track error exception.*)
		Inlet01HomeException : BOOL; (*Inlet01 home exception.*)
		Inlet01TorqueException : BOOL; (*Inlet01 torque exception.*)
		Inlet01DriveException : BOOL; (*Inlet01 drive exception.*)
		Inlet01TemperatureError : BOOL; (*Inlet01 temperature exception.*)
		Inlet01SafetyException : BOOL; (*Inlet01 safety exception.*)
		Inlet01NotInOpException : BOOL; (*Inlet01 not in operational exception.*)
		Inlet02TrackException : BOOL; (*Inlet02 track error exception.*)
		Inlet02HomeException : BOOL; (*Inlet02 home exception.*)
		Inlet02TorqueException : BOOL; (*Inlet02 torque exception.*)
		Inlet02DriveException : BOOL; (*Inlet02 drive exception.*)
		Inlet02TemperatureError : BOOL; (*Inlet02 temperature exception.*)
		Inlet02SafetyException : BOOL; (*Inlet02 safety exception.*)
		Inlet02NotInOpException : BOOL; (*Inlet02 not in operational exception.*)
		Inlet03TrackException : BOOL; (*Inlet03 track error exception.*)
		Inlet03HomeException : BOOL; (*Inlet03 home exception.*)
		Inlet03TorqueException : BOOL; (*Inlet03 torque exception.*)
		Inlet03DriveException : BOOL; (*Inlet03 drive exception.*)
		Inlet03TemperatureError : BOOL; (*Inlet03 temperature exception.*)
		Inlet03SafetyException : BOOL; (*Inlet03 safety exception.*)
		Inlet03NotInOpException : BOOL; (*Inlet03 not in operational exception.*)
		Inlet04TrackException : BOOL; (*Inlet04 track error exception.*)
		Inlet04HomeException : BOOL; (*Inlet04 home exception.*)
		Inlet04TorqueException : BOOL; (*Inlet04 torque exception.*)
		Inlet04DriveException : BOOL; (*Inlet04 drive exception.*)
		Inlet04TemperatureError : BOOL; (*Inlet04 temperature exception.*)
		Inlet04SafetyException : BOOL; (*Inlet04 safety exception.*)
		Inlet04NotInOpException : BOOL; (*Inlet04 not in operational exception.*)
		Inlet05TrackException : BOOL; (*Inlet05 track error exception.*)
		Inlet05HomeException : BOOL; (*Inlet05 home exception.*)
		Inlet05TorqueException : BOOL; (*Inlet05 torque exception.*)
		Inlet05DriveException : BOOL; (*Inlet05 drive exception.*)
		Inlet05TemperatureError : BOOL; (*Inlet05 temperature exception.*)
		Inlet05SafetyException : BOOL; (*Inlet05 safety exception.*)
		Inlet05NotInOpException : BOOL; (*Inlet05 not in operational exception.*)
		Inlet06TrackException : BOOL; (*Inlet06 track error exception.*)
		Inlet06HomeException : BOOL; (*Inlet06 home exception.*)
		Inlet06TorqueException : BOOL; (*Inlet06 torque exception.*)
		Inlet06DriveException : BOOL; (*Inlet06 drive exception.*)
		Inlet06TemperatureError : BOOL; (*Inlet06 temperature exception.*)
		Inlet06SafetyException : BOOL; (*Inlet06 safety exception.*)
		Inlet06NotInOpException : BOOL; (*Inlet06 not in operational exception.*)
		Inlet07TrackException : BOOL; (*Inlet07 track error exception.*)
		Inlet07HomeException : BOOL; (*Inlet07 home exception.*)
		Inlet07TorqueException : BOOL; (*Inlet07 torque exception.*)
		Inlet07DriveException : BOOL; (*Inlet07 drive exception.*)
		Inlet07TemperatureError : BOOL; (*Inlet07 temperature exception.*)
		Inlet07SafetyException : BOOL; (*Inlet07 safety exception.*)
		Inlet07NotInOpException : BOOL; (*Inlet07 not in operational exception.*)
		Inlet08TrackException : BOOL; (*Inlet08 track error exception.*)
		Inlet08HomeException : BOOL; (*Inlet08 home exception.*)
		Inlet08TorqueException : BOOL; (*Inlet08 torque exception.*)
		Inlet08DriveException : BOOL; (*Inlet08 drive exception.*)
		Inlet08TemperatureError : BOOL; (*Inlet08 temperature exception.*)
		Inlet08SafetyException : BOOL; (*Inlet08 safety exception.*)
		Inlet08NotInOpException : BOOL; (*Inlet08 not in operational exception.*)
		Inlet09TrackException : BOOL; (*Inlet09 track error exception.*)
		Inlet09HomeException : BOOL; (*Inlet09 home exception.*)
		Inlet09TorqueException : BOOL; (*Inlet09 torque exception.*)
		Inlet09DriveException : BOOL; (*Inlet09 drive exception.*)
		Inlet09TemperatureError : BOOL; (*Inlet09 temperature exception.*)
		Inlet09SafetyException : BOOL; (*Inlet09 safety exception.*)
		Inlet09NotInOpException : BOOL; (*Inlet09 not in operational exception.*)
		Inlet10TrackException : BOOL; (*Inlet10 track error exception.*)
		Inlet10HomeException : BOOL; (*Inlet10 home exception.*)
		Inlet10TorqueException : BOOL; (*Inlet10 torque exception.*)
		Inlet10DriveException : BOOL; (*Inlet10 drive exception.*)
		Inlet10TemperatureError : BOOL; (*Inlet10 temperature exception.*)
		Inlet10SafetyException : BOOL; (*Inlet10 safety exception.*)
		Inlet10NotInOpException : BOOL; (*Inlet10 not in operational exception.*)
		CarouselTrackException : BOOL; (*Carousel track error exception.*)
		CarouselHomeException : BOOL; (*Carousel home exception.*)
		CarouselTorqueException : BOOL; (*Carousel torque exception.*)
		CarouselDriveException : BOOL; (*Carousel drive exception.*)
		CarouselTemperatureError : BOOL; (*Carousel temperature exception.*)
		CarouselSafetyException : BOOL; (*Carousel safety exception.*)
		CarouselNotInOpException : BOOL; (*Carousel not in operational exception.*)
		Outlet01TrackException : BOOL; (*Outlet01 track error exception.*)
		Outlet01HomeException : BOOL; (*Outlet01 home exception.*)
		Outlet01TorqueException : BOOL; (*Outlet01 torque exception.*)
		Outlet01DriveException : BOOL; (*Outlet01 drive exception.*)
		Outlet01TemperatureError : BOOL; (*Outlet01 temperature exception.*)
		Outlet01SafetyException : BOOL; (*Outlet01 safety exception.*)
		Outlet01NotInOpException : BOOL; (*Outlet01 not in operational exception.*)
		Outlet02TrackException : BOOL; (*Outlet02 track error exception.*)
		Outlet02HomeException : BOOL; (*Outlet02 home exception.*)
		Outlet02TorqueException : BOOL; (*Outlet02 torque exception.*)
		Outlet02DriveException : BOOL; (*Outlet02 drive exception.*)
		Outlet02TemperatureError : BOOL; (*Outlet02 temperature exception.*)
		Outlet02SafetyException : BOOL; (*Outlet02 safety exception.*)
		Outlet02NotInOpException : BOOL; (*Outlet02 not in operational exception.*)
		Outlet03TrackException : BOOL; (*Outlet03 track error exception.*)
		Outlet03HomeException : BOOL; (*Outlet03 home exception.*)
		Outlet03TorqueException : BOOL; (*Outlet03 torque exception.*)
		Outlet03DriveException : BOOL; (*Outlet03 drive exception.*)
		Outlet03TemperatureError : BOOL; (*Outlet03 temperature exception.*)
		Outlet03SafetyException : BOOL; (*Outlet03 safety exception.*)
		Outlet03NotInOpException : BOOL; (*Outlet03 not in operational exception.*)
		Outlet04TrackException : BOOL; (*Outlet04 track error exception.*)
		Outlet04HomeException : BOOL; (*Outlet04 home exception.*)
		Outlet04TorqueException : BOOL; (*Outlet04 torque exception.*)
		Outlet04DriveException : BOOL; (*Outlet04 drive exception.*)
		Outlet04TemperatureError : BOOL; (*Outlet04 temperature exception.*)
		Outlet04SafetyException : BOOL; (*Outlet04 safety exception.*)
		Outlet04NotInOpException : BOOL; (*Outlet04 not in operational exception.*)
		Outlet05TrackException : BOOL; (*Outlet05 track error exception.*)
		Outlet05HomeException : BOOL; (*Outlet05 home exception.*)
		Outlet05TorqueException : BOOL; (*Outlet05 torque exception.*)
		Outlet05DriveException : BOOL; (*Outlet05 drive exception.*)
		Outlet05TemperatureError : BOOL; (*Outlet05 temperature exception.*)
		Outlet05SafetyException : BOOL; (*Outlet05 safety exception.*)
		Outlet05NotInOpException : BOOL; (*Outlet05 not in operational exception.*)
		Outlet06TrackException : BOOL; (*Outlet06 track error exception.*)
		Outlet06HomeException : BOOL; (*Outlet06 home exception.*)
		Outlet06TorqueException : BOOL; (*Outlet06 torque exception.*)
		Outlet06DriveException : BOOL; (*Outlet06 drive exception.*)
		Outlet06TemperatureError : BOOL; (*Outlet06 temperature exception.*)
		Outlet06SafetyException : BOOL; (*Outlet06 safety exception.*)
		Outlet06NotInOpException : BOOL; (*Outlet06 not in operational exception.*)
	END_STRUCT;
END_TYPE

(*Outlet module*)

TYPE
	ST_OutletInterface : 	STRUCT  (*Outlet module input/output interface structure*)
		Commands : ST_OutletCommands; (*Outlet commands structure*)
		Parameters : ST_OutletParameters; (*Outlet parameters structure*)
		Status : ST_OutletStatus; (*Outlet status structure*)
		Exceptions : ST_OutletExceptions; (*Outlet  exceptions structure*)
	END_STRUCT;
	ST_OutletCommands : 	STRUCT  (*Outlet module commands structure*)
		AutoOutletModule : BOOL; (*Auto modality request for auto module in multi mode.*)
		JogOutletModule : BOOL; (*Jog modality request for auto module in multi mode.*)
		QuickStopOutletModule : BOOL; (*Quick stop on Outlet module; quick stop not active signal 1.*)
		StartOutletModule : BOOL; (*Start on Outlet module.*)
		JogPushButtonOutletModule : BOOL; (*Jog push button for Outlet module.*)
		SlowMotionBackward : BOOL; (*Slow motion backward on Outlet module.*)
		SlowMotionForward : BOOL; (*Slow motion forward on Outlet module.*)
		AbsolutePositionSensor : BOOL;
		VelocityAxisStop : BOOL;
	END_STRUCT;
	ST_OutletStatus : 	STRUCT  (*Outlet module status structure*)
		ModuleHomed : BOOL; (*Outlet Module Homed; all axes are homed.*)
		ModuleInPosition : BOOL; (*Outlet Module In Position; all axes are standstill and in position.*)
		ModuleRunning : BOOL; (*Outlet Module Running; at least one axis is not standstill.*)
		ModulePowered : BOOL; (*Outlet Module Powered; Outlet module is enabled from a safety point of view.*)
		EnableAutoModality : BOOL; (*Outlet Module Enable Auto Modality; during machine multi mode all condition are valid for enabling the Auto modality.*)
		EnableJogModality : BOOL; (*Outlet Module Enable Auto Modality; during machine multi mode all condition are valid for enabling the Jog modality.*)
		ModuleJogActive : BOOL; (*Outlet Module Jog Active; the jog modality on the Outlet module is active.*)
		AutoActive : BOOL; (*Outlet Module Auto Active; the auto modality on the Outlet module is active.*)
		SlowMotionActive : BOOL; (*Outlet Module Slow Motion Active; the slow motion on the Outlet module is active.*)
		JogCmdFeedback : BOOL; (*Outlet Module Jog Command Feedback.*)
		AutoCmdFeedback : BOOL; (*Outlet Module Auto Command Feedback.*)
		ModuleNotInitialized : BOOL; (*Outlet Module Not Initialized; the Outlet module isn't initialized. PowerOn the module.*)
		ModuleReal : BOOL; (*Outlet Module Real; at least one axis is real on the Outlet module.*)
		MainAxisReal : BOOL; (*Main axis on filler module is real.*)
		Out01Real : BOOL; (*Axis Outlet01 on filler module is real.*)
		Out02Real : BOOL; (*Axis Outlet02 on filler module is real.*)
		Out03Real : BOOL; (*Axis Outlet03 on filler module is real.*)
		Out04Real : BOOL; (*Axis Outlet04 on filler module is real.*)
		Out05Real : BOOL; (*Axis Outlet05 on filler module is real.*)
		Out06Real : BOOL; (*Axis Outlet06 on filler module is real.*)
		Velocity : REAL; (*Outlet module actual velocity [bph]*)
		AbsolutePosition : LREAL;
		AbsolutePositionValid : BOOL;
	END_STRUCT;
	ST_OutletParameters : 	STRUCT  (*Outlet module parameters structure*)
		AutoSpeedOutletModule : REAL; (*Auto speed for Outlet module [bph].*)
		AbsolutePositionValveOffset : UINT;
		ConveyorKs : REAL;
		WheelValvesNumber : UINT;
		TorqueError : CFG_FillerTorque_Type;
	END_STRUCT;
	ST_OutletExceptions : 	STRUCT  (*Outlet module exception structure*)
		MainAxisTrackException : BOOL; (*Main Axis Outlet module track error exception.*)
		MainAxisHomeException : BOOL; (*Main Axis Outlet module home exception.*)
		MainAxisTorqueException : BOOL; (*Main Axis Outlet module torque exception.*)
		MainAxisDriveException : BOOL; (*Main Axis Outlet module drive exception.*)
		MainAxisTemperatureError : BOOL; (*Main Axis Outlet module temperature exception.*)
		MainAxisSafetyException : BOOL; (*Main Axis Outlet module safety exception.*)
		MainAxisNotInOpException : BOOL; (*Main Axis Outlet module not in operational exception.*)
		Outlet01TrackException : BOOL; (*Outlet01 track error exception.*)
		Outlet01HomeException : BOOL; (*Outlet01 home exception.*)
		Outlet01TorqueException : BOOL; (*Outlet01 torque exception.*)
		Outlet01DriveException : BOOL; (*Outlet01 drive exception.*)
		Outlet01TemperatureError : BOOL; (*Outlet01 temperature exception.*)
		Outlet01SafetyException : BOOL; (*Outlet01 safety exception.*)
		Outlet01NotInOpException : BOOL; (*Outlet01 not in operational exception.*)
		Outlet02TrackException : BOOL; (*Outlet02 track error exception.*)
		Outlet02HomeException : BOOL; (*Outlet02 home exception.*)
		Outlet02TorqueException : BOOL; (*Outlet02 torque exception.*)
		Outlet02DriveException : BOOL; (*Outlet02 drive exception.*)
		Outlet02TemperatureError : BOOL; (*Outlet02 temperature exception.*)
		Outlet02SafetyException : BOOL; (*Outlet02 safety exception.*)
		Outlet02NotInOpException : BOOL; (*Outlet02 not in operational exception.*)
		Outlet03TrackException : BOOL; (*Outlet03 track error exception.*)
		Outlet03HomeException : BOOL; (*Outlet03 home exception.*)
		Outlet03TorqueException : BOOL; (*Outlet03 torque exception.*)
		Outlet03DriveException : BOOL; (*Outlet03 drive exception.*)
		Outlet03TemperatureError : BOOL; (*Outlet03 temperature exception.*)
		Outlet03SafetyException : BOOL; (*Outlet03 safety exception.*)
		Outlet03NotInOpException : BOOL; (*Outlet03 not in operational exception.*)
		Outlet04TrackException : BOOL; (*Outlet04 track error exception.*)
		Outlet04HomeException : BOOL; (*Outlet04 home exception.*)
		Outlet04TorqueException : BOOL; (*Outlet04 torque exception.*)
		Outlet04DriveException : BOOL; (*Outlet04 drive exception.*)
		Outlet04TemperatureError : BOOL; (*Outlet04 temperature exception.*)
		Outlet04SafetyException : BOOL; (*Outlet04 safety exception.*)
		Outlet04NotInOpException : BOOL; (*Outlet04 not in operational exception.*)
		Outlet05TrackException : BOOL; (*Outlet05 track error exception.*)
		Outlet05HomeException : BOOL; (*Outlet05 home exception.*)
		Outlet05TorqueException : BOOL; (*Outlet05 torque exception.*)
		Outlet05DriveException : BOOL; (*Outlet05 drive exception.*)
		Outlet05TemperatureError : BOOL; (*Outlet05 temperature exception.*)
		Outlet05SafetyException : BOOL; (*Outlet05 safety exception.*)
		Outlet05NotInOpException : BOOL; (*Outlet05 not in operational exception.*)
		Outlet06TrackException : BOOL; (*Outlet06 track error exception.*)
		Outlet06HomeException : BOOL; (*Outlet06 home exception.*)
		Outlet06TorqueException : BOOL; (*Outlet06 torque exception.*)
		Outlet06DriveException : BOOL; (*Outlet06 drive exception.*)
		Outlet06TemperatureError : BOOL; (*Outlet06 temperature exception.*)
		Outlet06SafetyException : BOOL; (*Outlet06 safety exception.*)
		Outlet06NotInOpException : BOOL; (*Outlet06 not in operational exception.*)
	END_STRUCT;
END_TYPE

(*Filler Module Safety Interface*)

TYPE
	ST_FillerSafetyInterface : 	STRUCT  (*Filler module input/output safety interface structure*)
		Commands : ST_FillerSafetyCommands; (*Filler safety commands*)
		Status : ST_FillerSafetyStatus; (*Filler safety status*)
	END_STRUCT;
	ST_FillerSafetyCommands : 	STRUCT  (*Filler safety commands*)
		EnableModule : BOOL; (*Hardware enable of Filler Module*)
		AxesDiag : ARRAY[0..CST_LastFillerModuleAxis]OF ST_AxesDiag; (*Diagnostic datapoints for filler module axes*)
	END_STRUCT;
	ST_FillerSafetyStatus : 	STRUCT  (*Filler safety status*)
		ModulePowered : BOOL; (*Filler Module Powered*)
	END_STRUCT;
END_TYPE

(*Inlet Module Safety Interface*)

TYPE
	ST_InletSafetyInterface : 	STRUCT  (*Inlet module input/output safety interface structure*)
		Commands : ST_InletSafetyCommands; (*Inlet safety commands*)
		Status : ST_InletSafetyStatus; (*Inlet safety status*)
	END_STRUCT;
	ST_InletSafetyCommands : 	STRUCT  (*Inlet safety commands*)
		EnableModule : BOOL; (*Hardware enable of inlet module*)
		AxesDiag : ARRAY[0..CST_LastInletModuleAxis]OF ST_AxesDiag; (*Diagnostic datapoints for filler module axes*)
	END_STRUCT;
	ST_InletSafetyStatus : 	STRUCT  (*Inlet safety status
*)
		ModulePowered : BOOL; (*Inlet Module Powered*)
	END_STRUCT;
END_TYPE

(*Outlet Module Safety Interface*)

TYPE
	ST_OutletSafetyInterface : 	STRUCT  (*Outlet module input/output safety interface structure*)
		Commands : ST_OutletSafetyCommands; (*Outlet safety commands
*)
		Status : ST_OutletSafetyStatus; (*Outlet safety status*)
	END_STRUCT;
	ST_OutletSafetyCommands : 	STRUCT  (*Outlet safety commands
*)
		EnableModule : BOOL; (*Hardware enable of outlet module*)
		AxesDiag : ARRAY[0..CST_LastOutletModuleAxis]OF ST_AxesDiag; (*Diagnostic datapoints for filler module axes*)
	END_STRUCT;
	ST_OutletSafetyStatus : 	STRUCT  (*Outlet safety status*)
		ModulePowered : BOOL; (*Outlet Module Powered*)
	END_STRUCT;
END_TYPE

(*Axes Diag Safety Struct*)

TYPE
	ST_AxesDiag : 	STRUCT  (*Structure to be connected directly to Hardware*)
		DI_SafeModuleOK : BOOL; (*Safe Module OK Digital input*)
		DI_STOActive : BOOL; (*Safe Torque Off functionality is active*)
		DI_STO1Active : BOOL; (*Safe Torque Off 1 Active*)
		DI_SOSActive : BOOL; (*Safe Operating Stop is active*)
		DI_SS1Active : BOOL; (*Safe Stop 1 is active*)
		DI_SS2Active : BOOL; (*Safe Stop 2 is active*)
		DI_SLS1Active : BOOL; (*Safe Limited speed 1*)
		DI_Operational : BOOL; (*Drive in operational state*)
		DI_NotErrENC : BOOL; (*Encoder not in error state*)
		DI_NotErrFUNC : BOOL; (*Drive not in functional error*)
	END_STRUCT;
END_TYPE

(*MOTION*)

TYPE
	MC_Type : 	STRUCT
		DataOut : MC_DataOut_Type;
	END_STRUCT;
	MC_DataOut_Type : 	STRUCT
		MachineRunning : BOOL;
		ActualSpeed : REAL;
		MaxSpeed : REAL;
	END_STRUCT;
END_TYPE
```

### MNM_Global.typ
```iecst
(*MAIN DRIVE CONTROL*)

TYPE
	MNM_Type : 	STRUCT
		DataOut : MNM_DataOut_Type;
	END_STRUCT;
	MNM_DataOut_Type : 	STRUCT
		HornFlrRequest : BOOL;
		StartLightBlinkRequest : BOOL;
		StartLightFixRequest : BOOL;
		CopSpeedReqReached : BOOL;
		RnsSpeedReqReached : BOOL;
		CapSpeedReqReached : BOOL;
		DmcSpeedReqReached : BOOL;
		SftSpeedReqReached : BOOL;
		SkidSpeedReqReached : BOOL;
		EmptySpeedReached : BOOL;
		ContBlockSpeedReached : BOOL;
		ContBlock1Requested : BOOL;
		ContBlock2Requested : BOOL;
		MachineRunning : BOOL; (*Module Running*)
		ReadyForVortexCalib : BOOL;
		ReadyForCoupling : BOOL;
		PartnerReadyToRun : BOOL;
		OperatorPresence : BOOL;
		FixSpeedRequest : BOOL;
		OutletSpeed : REAL;
		LackInlet1 : BOOL;
		LackInlet2 : BOOL;
		COPInletContBlockSpeedReached : BOOL;
		ContainerStop : BOOL;
		DesyncroRequest : BOOL;
		CapperPositioningDone : BOOL;
		SingleAxisInPosition : BOOL;
		RinserAxisDisabled : BOOL;
		DoserAxisDisabled : BOOL;
		FillerAxisDisabled : BOOL;
		FillingValvePositioningDone : BOOL;
		ReversePositioningDone : BOOL;
		DmcPositioningDone : BOOL;
		PhaseDone : BOOL;
		ConfigReqLoaded : BOOL;
		StartRequest : BOOL;
		InletSpeed : REAL;
	END_STRUCT;
END_TYPE
```

### MNT_Global.typ
```iecst
(*MAINTENANCE*)

TYPE
	MNT_Type : 	STRUCT  (*v1.4*)
		DataOut : MNT_DataOut_Type;
	END_STRUCT;
	MNT_DataOut_Type : 	STRUCT  (*v1.4*)
		LotoInExecution : BOOL;
		LotoValvesOpening : BOOL;
		LotoAirDischarge : BOOL;
		LotoAirDischargePilot : BOOL;
		LotoDmcOn : BOOL;
		LotoStep : USINT;
		LotoDevices : INT;
	END_STRUCT;
END_TYPE
```

### OPS_Global.typ
```iecst
(*SAFETY*)

TYPE
	OPS_Type : 	STRUCT
		DataOut : OPS_DataOut_Type; (*SAFE_PLC Inputs*)
	END_STRUCT;
	OPS_DataOut_Type : 	STRUCT
		EmergencyOk : BOOL := TRUE;
		FlrDoorsOk : BOOL := TRUE;
		DoorsOk : BOOL;
		GeneralAirOn : BOOL;
		ConfinementZoneRed : BOOL;
		BeaconHornJog : BOOL; (*Blow horn request for jog*)
		FlrModeSelectorAuto : BOOL := TRUE;
		FlrModeSelectorAdjustment : BOOL := TRUE;
		FlrModeSelectorJog : BOOL := TRUE;
		JogStartPb : BOOL := TRUE;
		SelModeChange : BOOL; (*Mode selection Error*)
		EnableDrive : BOOL;
		EnablePump : BOOL;
		EnableProcessValves : BOOL;
		EnableCopValves : BOOL; (*V4.A.A.1.6.11a*)
		EnableVerticalDrive : BOOL; (*V4.A.A.1.6.6*)
		BufferDoorOpened : BOOL;
		BufferDoorFault : BOOL;
		HMIDoorUnlock : BOOL;
		LabellerTrasferDoorOpenRequest : BOOL;
		BlowerTrasferDoorOpenRequest : BOOL;
		ActisTrasferDoorOpenRequest : BOOL; (*V4.A.A.1.6.12*)
		LabellerTrasferGateOpened : BOOL;
		BlowerTrasferGateOpened : BOOL;
		ActisTrasferGateOpened : BOOL; (*V4.A.A.1.6.12*)
		AutomaticInletGate : BOOL; (*Not Used in Glass Machine*)
		InletGateOpened : BOOL; (*V4.A.A.1.6.12h*)
		InletGateClosed : BOOL;
		OutletGateClosed : BOOL;
		OutletGateOpened : BOOL; (*V4.A.A.1.7.0*)
		OperatorPresence : BOOL;
		ContainerStop : BOOL; (*//1.63*)
		ConfigSaveReq : BOOL;
		FlrLiftingEnabled : BOOL;
		FillerLiftPw : BOOL; (*maste nuovo*)
		FillerLiftPwFault : BOOL; (*master nuovo*)
		DoorsOpenExceptGloves : BOOL; (*V4.A.A.1.7.0*)
	END_STRUCT;
END_TYPE
```

### REL_Global.typ
```iecst
(*ELECTRONIC FUSES*)

TYPE
	REL_Type : 	STRUCT
		DataOut : REL_DataOut_Type;
	END_STRUCT;
	REL_DataOut_Type : 	STRUCT
		ElectronicFusesPresence : BOOL;
		GlobalPowerOn : BOOL := TRUE;
		Station : ARRAY[1..16]OF REL_Channel_Type;
	END_STRUCT;
	REL_Channel_Type : 	STRUCT
		Ch : ARRAY[1..16]OF REL_Status_Type;
	END_STRUCT;
	REL_Status_Type : 	STRUCT
		ConfigurationError : BOOL;
		PoweredOn : BOOL;
		Overload : BOOL;
		ShortCircuit : BOOL;
	END_STRUCT;
END_TYPE
```

### RCP_Global.typ
```iecst
(*PRODUCTION RECIPE MANAGER*)

TYPE
	RCP_Type : 	STRUCT
		DataOut : RCP_DataOut_Type;
	END_STRUCT;
	RCP_DataOut_Type : 	STRUCT
		RecipeDownload : BOOL;
		RecipeDownloaded : BOOL;
	END_STRUCT;
END_TYPE
```

### SFT_Global.typ
```iecst
(*CONTAINERS SHIFT REGISTER*)

TYPE
	SFT_Type : 	STRUCT
		DataOut : SFT_DataOut_Type;
	END_STRUCT;
	SFT_DataOut_Type : 	STRUCT
		Alarm : SFT_Alarm_Type;
		ContainersBlock1 : BOOL; (*Block container in corrispondence of FV disable*)
		ContainersBlock2 : BOOL; (*Block container in corrispondence of FV disable*)
		ContainerStop : BOOL; (*//1.63*)
		ContainersReleaseEarlier1 : BOOL;
		ContainersReleaseEarlier2 : BOOL;
		ContainersAtCarouselOutlet : BOOL;
		ContainerAtMachineOutlet : BOOL;
		CombiEmpty : BOOL; (*No containers in the combi*)
		MachineEmpty : BOOL; (*No containers in the machine*)
		_20Bottles_AtExit : BOOL; (*Signals For Conveyor - Information 20 bottles at machine exit*)
		RinserTreatmentRequest : BOOL;
		BottleCoolingRequest : BOOL;
		InletConveyorEmpty : BOOL;
		OutletConveyorEmpty : BOOL;
		CapsAirRequest : BOOL; (*Closing Unit - Air Blow*)
		CapsReleaseProductionReady : BOOL;
		CapsReleaseEmptyingReady : BOOL;
		CapsReleaseEmpty : BOOL; (*v1.5*)
		CappingHeadAtMachineGetData : BOOL; (*V4.A.A.1.6.12*)
		CapOnCappingHead : BOOL; (*v1.5*)
		FMC_PreClosingContainerReq : BOOL;
		FMC_ContainerPresenceReq : BOOL;
		FMC_WashCenteringCup : BOOL;
		FMC_StartFillingReq : BOOL;
		FillingValveRinseReq : BOOL;
		ManPreformLoadingReq : BOOL;
		VBS_Presence : BOOL;
		DmcNotInserted : BOOL;
		DmcNotRemoved : BOOL;
		CounterDone : BOOL;
		ValveDisabledPreformBlock : BOOL;
		ValveDisabledLbrBottleEjection : BOOL;
		SlowDownContBlockReq : BOOL;
		ContBlockSpeedReq : BOOL;
		ManualContainersReleaseEnable : BOOL; (*Block container in corrispondence of FV disable*)
		OutletShowerReq : BOOL;
		NeckRinseReq : BOOL;
		MachineInletStatus : BOOL;
		COPInletContSlowSpeedReq : BOOL;
		COPInletContConvEmptyRunning : BOOL;
		COPInletContConvEmptyDone : BOOL;
		FillingValvePositionReq : BOOL; (*Filling valve positioning request*)
		PreformManualLoading : BOOL; (*v1.6*)
		CapTreatmentStart : BOOL; (*V4.A.A.1.7.0*)
		NoBottleNoSprayPistonFault : BOOL; (*vrma*)
		NoBottleNoSprayActive : BOOL; (*vrma*)
		FirstHalfDmcInsered : BOOL;
		SecondHalfCounterDone : BOOL;
		SecondHalfDmcNotInserted : BOOL;
		SecondHalfDmcNotRemoved : BOOL;
		FillingValveAtMachineInlet : INT;
		CappingHeadAtMachineInlet : INT;
		CapHeadNumberInTangency : INT; (*V4.A.A.1.6.12*)
		RinsingNozzleAtMachineInlet : INT; (*V4.A.A.1.6.12*)
		RinserBypassedPointer : INT; (*V4.A.A.1.6.12*)
		BottleBurstWashRampActivation : ARRAY[1..3]OF BOOL; (*master nuovo*)
		FoamerRequest : BOOL;
		CrownsReleaseProductionReady : BOOL;
		CrownsAirRequest : BOOL;
		FillingValve1 : BOOL; (*FCI:TEST v1.7.4a*)
		CapperHead1 : BOOL; (*FCI:TEST v1.7.4a*)
		CrownerHead1 : BOOL; (*FCI:TEST v1.7.4a*)
		DoserHead1 : BOOL; (*v999hema*)
		AuxBlowerMold1 : BOOL; (*FCI:TEST v1.7.4a*)
		AuxLabelerPlate1 : BOOL; (*FCI:TEST v1.7.4a*)
		ContainersInFiller : UINT; (*Number of containers in the machine*)
		ContainersInConveyorReject : UINT; (*Number of container to be reject after COP vrmaCOP *)
		ContainersInMachine : UINT; (*Number of containers in the machine*)
		ContainersToFillFillerOnly : UINT;
		ContainersToFill : UINT; (*Number of containers to be filled (From Container Block To Inlet Tangency)*)
		ContainersToCap : UINT; (*Number of containers to be filled (From Container Block To Inlet Tangency) V4.A.A.1.7.0*)
		BottleCoolingFillerSteps : UINT;
		RinserFillerSteps : UINT; (*V4.A.A.1.6.12*)
		DoserFillerSteps : UINT; (*v999hema*)
		NumberDmcInserted : UINT;
		FillingValvePosValue : UINT; (*Number of filling valve to position in the ispection point*)
		CopPurgeStep : UINT; (*vrmaCOP*)
		ContBlockSpeedValue : REAL;
		COPInletContBlockSpeedValue : REAL;
		FMC_PreClosingContainerReqByte : USINT; (*v1.7.4*)
		FMC_ContainerPresenceReqByte : USINT; (*v1.7.4*)
		FMC_StartFillingReqByte : USINT; (*v1.7.4*)
		DmcClockSensorBroken : BOOL;
		ChannelEmptyingDone : BOOL; (*vrmaCOP*)
	END_STRUCT;
	SFT_Alarm_Type : 	STRUCT
		BottMissingForFillerFault : BOOL;
		Category : DINT;
		ID : DINT;
		OmacCode : DINT;
	END_STRUCT;
END_TYPE

(*SHIFT*)

TYPE
	MachineShift_Type : 	STRUCT
		ShiftInfo : UINT;
		FillingNozzle : USINT;
		CrownerHead : USINT;
		DoserHead : USINT; (*v999hema*)
		CappingHead : USINT;
		RinsingNozzle : USINT; (*V4.A.A.1.7.0*)
	END_STRUCT;
	CombiShift_Type : 	STRUCT
		MoldNumber : UINT; (*V1.61*)
		CombiInfo : UINT;
		AlarmId : UDINT;
		Category : UDINT;
		OmacCode : UDINT;
	END_STRUCT;
END_TYPE
```

### TNK_Global.typ
```iecst
(*TANK*)

TYPE
	TNK_Type : 	STRUCT
		DataOut : TNK_DataOut_Type;
	END_STRUCT;
	TNK_DataOut_Type : 	STRUCT
		Wait : BOOL;
		CipMode : BOOL;
		CipDrainMode : BOOL;
		RinseMode : BOOL;
		DrainMode : BOOL;
		ProdMode : BOOL;
		PushBackMode : BOOL;
		StartUp : BOOL;
		SipMode : BOOL;
		DeEnergization : BOOL;
		EndProduction : BOOL;
		Calibration : BOOL; (*V4.A.A.1.6.13*)
		ContainerStop : BOOL; (*//1.63*)
		DummyContainersIns : BOOL;
		DummyContainersDis : BOOL;
		CopInProductionActive : BOOL;
		StartUpHOT : BOOL;
		StartCipRinser : BOOL;
		APCORunning : BOOL;
		DisableCipRinser : BOOL;
	END_STRUCT;
END_TYPE
```

### DOS_Global.typ
```iecst
(*FLAVOR DOSER*)

TYPE
	DOS_Type : 	STRUCT
		DataOut : DOS_DataOut_Type;
	END_STRUCT;
	DOS_DataOut_Type : 	STRUCT  (*v999hema*)
		FillingHeatingProd : BOOL;
		FillingProd : BOOL;
		WaitMode : BOOL;
		ProdMode : BOOL;
		ProductRequest : BOOL;
		ProductionEnd : BOOL;
		ReadyForHeating : BOOL;
		DoserFull : BOOL;
		AVJ201Open : BOOL;
		DoserEmpty : BOOL;
		DoserInTemperature : BOOL;
		RecoveryEnd : BOOL;
		EjectionRequest : BOOL;
		HotWaterReq : BOOL;
		NecessaryBottleEndProd : REAL;
		CipMode : BOOL;
		CipConditionOk : BOOL;
		CipSolutionReq : BOOL;
		CipRecovery : BOOL;
		CipRecoveryEnd : BOOL;
		CipAlarm : BOOL;
		RinseEnd : BOOL;
		RinseReq : BOOL;
		CipDrainEnd : BOOL;
		CipLevelReached : BOOL;
		CipSystemFlooded : BOOL;
		RinseAfterProdReq : BOOL;
		RinseMode : BOOL;
		RinseAfterProdEnd : BOOL;
		DrainMode : BOOL;
		CopMode : BOOL;
		CopAfterCipReq : BOOL;
		CopRunning : BOOL;
		AromePodReq : BOOL;
		MachineStart : BOOL;
		MachineStop : BOOL;
		DoserExcluded : BOOL;
		DoserIncluded : BOOL;
		ByPassed : BOOL;
		AxisEnableRequest : BOOL;
		AxisDisableRequest : BOOL;
		FillerAxisDisableRequest : BOOL;
		StepCounterRequest : BOOL;
		FixSpeedRequest : BOOL;
		PositionReached : BOOL;
		CommandToValve : BOOL;
		FixSpeedValue : REAL;
		FillerProdStartEnable : BOOL;
		FillerCipStartEnable : BOOL;
		FillerRinseStartEnable : BOOL;
		PhasingWithDos : BOOL;
		PhasingWithoutDos : BOOL;
	END_STRUCT;
END_TYPE
```

### Sequencer.typ
```iecst
(*SEQUENCER PERMANENT TYPE*)

TYPE
	SEQ_Permanent_Type : 	STRUCT
		SeqActualStep : UINT;
		SeqBackupStep : UINT;
		SeqMode1 : UINT;
		SeqMode2 : UINT;
		SeqAuxiliary : UINT;
	END_STRUCT;
END_TYPE
```

### BTC_Global.typ - not listed in the package file held
```iecst
(*BOTTLE BOTTOM COOLING*)

TYPE
	BTC_Type : 	STRUCT
		DataOut : BTC_DataOut_Type;
	END_STRUCT;
	BTC_DataOut_Type : 	STRUCT
		Idle : BOOL; (*v1.4*)
		StepCountReq : BOOL;
		CipMode : BOOL;
		CipDrainMode : BOOL;
		RinseMode : BOOL;
		DrainMode : BOOL;
		ProdMode : BOOL;
		StartUp : BOOL;
		CopMode : BOOL;
		DeEnergization : BOOL;
		SamplingCommand : BOOL; (*V4.A.A.1.6.12*)
		SamplingInPosition : BOOL; (*V4.A.A.1.6.12*)
		ContainerStop : BOOL; (*//1.63*)
		WaterFlow : REAL;
		Temperature : REAL;
		TemperatureGlicol : REAL; (*V4.A.A.1.7.1*)
	END_STRUCT;
END_TYPE
```

### EIT_Global.typ - not listed in the package file held
```iecst
(*OPC VARIABLES - CHANGE THEM REQUIRES TO CHANGE OPC CONFIGURATION AND A WARM RESTART*)

TYPE
	EIT_Type : 	STRUCT
		Version : INT;
		Reason : DINT; (*Common - Reason code that stop the production on machine*)
		StopBit : BOOL; (*Common - Stop bit*)
		ProductionSpeed : REAL; (*Common - Production speed in CPM (Container per minute)*)
		SetSpeed : REAL; (*Common - Set speed*)
		UnitPerCount : INT; (*Common - Unit Per count*)
		SKU : INT; (*Common - SKU*)
		RecipeName : STRING[80]; (*Common - Recipe name*)
		OperatorPresence : BOOL; (*Common - Operator presence*)
		Format : STRING[20]; (*Common - Format*)
		MachineStatus : USINT; (*Common - Machine Status*)
		Count : EITCount_Type; (*Common - Specific Count tag different for each machine on the EITCount definition*)
		Measure : EITMeasure_Type; (*Common - Specific Measure tag different for each machine on the WITMeasure definition*)
		EZ : EITEZ_Type;
		SBO : EITSBO_Type;
		CapFeed : EITCapFeed_Type; (*Common - Uses for filler with Cap feeder*)
		Capper : EITCapper_Type; (*Common - Uses for filler with capper*)
		RunningEvent : EITRunningEvent_Type;
	END_STRUCT;
	EITCount_NotUsed_Type : 	STRUCT
		FillerRotationTotalizer : DINT; (*Filler - Number of filler revolution*)
		CapperRotationTotalizer : DINT; (*Filler - Number of capper revolution*)
		RinserRotationTotalizer : DINT; (*Filler - Number of rinser revolution*)
		BadFillingCount : DINT; (*Filler - Number of Bad filling count*)
		BadCappingCount : DINT; (*Filler - Number of Bad capping count*)
		BadRinsingCount : DINT; (*Filler - Number of Bad rinsing count*)
		ContainerOut : DINT; (*Filler - Count of container produced*)
		ContainerEjected : DINT; (*Filler - Count of container ejected*)
	END_STRUCT;
	EITCount_Type : 	STRUCT
		InfeedCount : UDINT; (*Filler - Count of infeed container on the machine*)
		ContainersBurstCount : UDINT; (*Filler - Number of Burst container count*)
		ContainersEjectManually : UDINT; (*Filler - Count of container ejected manually*)
		LowLevelEjectCount : UDINT;
		LPCA : UDINT; (*Filler - FlowLPCA V4.A.A.1.6.14k*)
		General_CO2 : UDINT;
		ClosingUnit_CO2 : UDINT;
		N2 : UDINT;
		ProcessWater : UDINT;
		CopWater : UDINT;
		BottleBottomCoolingWater : UDINT; (*V4.A.A.1.6.14k*)
		Product : UDINT;
		Steam : UDINT;
		FoodSteam : UDINT;
		ProductWater : UDINT; (*V4.A.A.1.6.14k*)
		Syrup : UDINT;
		ElectricalEnergy : UDINT; (*V4.A.A.1.6.14k*)
	END_STRUCT;
	EITMeasure_Type : 	STRUCT
		FlowLPCA : REAL; (*Filler - FlowLPCA V4.A.A.1.6.14k*)
		ElectricalPower : REAL; (*Filler - Electrical power KW*)
	END_STRUCT;
	EITEZ_Type : 	STRUCT
		StopBit : BOOL;
		Reason : INT;
	END_STRUCT;
	EITSBO_Type : 	STRUCT
		StopBit : BOOL;
		Reason : INT;
	END_STRUCT;
	EITCapFeed_Type : 	STRUCT
		StopBit : BOOL;
		Reason : INT;
	END_STRUCT;
	EITCapper_Type : 	STRUCT
		StopBit : BOOL;
		Reason : INT;
	END_STRUCT;
	EITRunningEvent_Type : 	STRUCT
		CapsLowLevel : BOOL;
		LidLowLevel : BOOL;
	END_STRUCT;
	EIT_ChangeOver_Type : 	STRUCT
		ToHLI : EIT_ChangeOver_To_Type;
		FromHLI : EIT_ChangeOver_From_Type;
	END_STRUCT;
	EIT_ChangeOver_From_Type : 	STRUCT
		NextProductReady : BOOL;
		PrepareForChange : BOOL;
		RinseRequested : BOOL;
		StopProduction : BOOL;
		WatchDog : INT;
		ProductToLoad : INT;
		NextRecipeId : UDINT;
		RemainingProdToDo : UDINT;
	END_STRUCT;
	EIT_ChangeOver_To_Type : 	STRUCT
		ChangeOverDone : BOOL;
		ChangeOverOptionOn : BOOL;
		ProductionEnded : BOOL;
		NextProductValidationRequest : BOOL;
		WatchDog : INT;
		ActualProduct : INT;
		ActualRecipeId : UDINT;
		ProductionBatchAvailable : UDINT;
	END_STRUCT;
	EIT_OMAC_Type : 	STRUCT
		Status : EIT_PMLs_Type;
		Command : EIT_PMLc_Type;
		Admin : EIT_PLMa_Type;
	END_STRUCT;
	EIT_PLMa_Type : 	STRUCT
		Alarm : EIT_PMLa_Alarm_Type;
	END_STRUCT;
	EIT_PMLa_Alarm_Type : 	STRUCT
		ID : UDINT;
		Value : UDINT;
		Message : STRING[80];
	END_STRUCT;
	EIT_PMLc_Type : 	STRUCT
		New_Member : USINT;
	END_STRUCT;
	EIT_PMLs_Type : 	STRUCT
		UnitModeCurrent : UDINT;
		StateCurrent : UDINT;
	END_STRUCT;
	WS_Type : 	STRUCT
		Communication : WS_Communication_Type;
		Tracking : WS_Tracking_Type;
		OperatingMode : WS_OperatingMode_Type;
		Omac : WS_Omac_Type;
		Fault : WS_Fault_Type;
		Pointer : WS_Pointer_Type;
		Parameter : WS_Parameter_Type;
		Counters : WS_Counters_Type;
	END_STRUCT;
	WS_Communication_Type : 	STRUCT
		WS_Error : UDINT; (*Tag-Number: 00000*)
		WS_PDACONT_Lenght : UDINT; (*Tag-Number: 00001*)
		WS_Test_Unsigned32_1 : UDINT; (*Tag-Number: 00011*)
		WS_Test_Unsigned32_2 : UDINT; (*Tag-Number: 00012*)
		WS_Test_Unsigned32_3 : UDINT; (*Tag-Number: 00013*)
		WS_Test_Signed32_1 : DINT; (*Tag-Number: 00014*)
		WS_Test_Signed32_2 : DINT; (*Tag-Number: 00015*)
		WS_Test_Signed32_3 : DINT; (*Tag-Number: 00016*)
		WS_Test_Real_1 : REAL; (*Tag-Number: 00017*)
		WS_Test_Real_2 : REAL; (*Tag-Number: 00018*)
		WS_Test_Real_3 : REAL; (*Tag-Number: 00019*)
		WS_Test_Hex32_1 : DWORD; (*Tag-Number: 00020*)
		WS_Test_Hex32_2 : DWORD; (*Tag-Number: 00021*)
		WS_Test_Hex32_3 : DWORD; (*Tag-Number: 00022*)
		WS_Test_String16_1 : STRING[1]; (*Tag-Number: 00023*)
		WS_Test_String16_2 : STRING[1]; (*Tag-Number: 00024*)
		WS_Test_String16_3 : STRING[1]; (*Tag-Number: 00025*)
	END_STRUCT;
	WS_Tracking_Type : 	STRUCT
		WS_Set_Batch_ID_L : DINT; (*Tag-Number: 00061*)
		WS_Set_Batch_ID_H : DINT; (*Tag-Number: 00062*)
		WS_Cur_Batch_ID_L : DINT; (*Tag-Number: 00063*)
		WS_Cur_Batch_ID_H : DINT; (*Tag-Number: 00064*)
	END_STRUCT;
	WS_OperatingMode_Type : 	STRUCT
		WS_Cur_Mode : UDINT; (*Tag-Number: 00100*)
		WS_Cur_Prog : UDINT; (*Tag-Number: 00200*)
		WS_Prog_Step : UDINT; (*Tag-Number: 00210*)
		WS_Cur_State : UDINT; (*Tag-Number: 00300*)
	END_STRUCT;
	WS_Omac_Type : 	STRUCT
		WS_Cur_Mach_Spd : REAL; (*Tag-Number: 00401*)
		WS_Set_Mach_Spd : REAL; (*Tag-Number: 00402*)
		WS_Mach_Design_Spd : REAL; (*Tag-Number: 00403*)
		WS_Mach_Cycle : UDINT; (*Tag-Number: 00501*)
		WS_Mat_Ready : DWORD; (*Tag-Number: 00601*)
		WS_Mat_Low : DWORD; (*Tag-Number: 00602*)
		WS_Prod_Ratio : UDINT; (*Tag-Number: 00701*)
	END_STRUCT;
	WS_Fault_Type : 	STRUCT
		WS_Not_Of_Fail_Code : UDINT; (*Tag-Number: 10000*)
	END_STRUCT;
	WS_Pointer_Type : 	STRUCT
		WS_Pointer_Code : UDINT; (*Tag-Number: 20000*)
	END_STRUCT;
	WS_Parameter_Type : 	STRUCT
		WS_Container_Type : UDINT; (*Tag-Number: 30003*)
		WS_Beer_Type : UDINT; (*Tag-Number: 30004*)
	END_STRUCT;
	WS_Measured_Type : 	STRUCT
		WS_Press_Bottling : REAL; (*Tag-Number: 40051*)
		WS_Temp_Bottling : REAL; (*Tag-Number: 40052*)
		WS_Temp_Product : REAL; (*Tag-Number: 40081*)
		WS_Cond_Product : REAL; (*Tag-Number: 40082*)
		WS_PH_Product : REAL; (*Tag-Number: 40083*)
		WS_O2_Product : REAL; (*Tag-Number: 40084*)
		WS_CO2_Product : REAL; (*Tag-Number: 40085*)
		WS_O_Press_Cleanroom : REAL; (*Tag-Number: 40121*)
	END_STRUCT;
	WS_Counters_Type : 	STRUCT
		WS_Tot_Containers : UDINT; (*Tag-Number: 50005*)
		WS_Good_Containers : UDINT; (*Tag-Number: 50006*)
		WS_Burst_Containers : UDINT; (*Tag-Number: 50009*)
		WS_Tot_Rej : UDINT; (*Tag-Number: 50011*)
	END_STRUCT;
END_TYPE
```

### ICO_Global.typ - not listed in the package file held
```iecst
(*INTELLI CHANGE OVER*)

TYPE
	ICO_Type : 	STRUCT
		DataOut : ICO_DataOut_Type;
	END_STRUCT;
	ICO_DataOut_Type : 	STRUCT
		ContainerStop : BOOL; (*//1.63*)
		Enabled : BOOL;
	END_STRUCT;
END_TYPE
```

### AID_Global.var
```iecst
VAR
	FB_GetTime : DTGetTime;
	FB_GetUtcTime : UtcDTGetTime;
	AID : AID_Type;
END_VAR
```

### CAP_Global.var
```iecst
VAR RETAIN
	VAR_CAP_ActualConfigEmptyValue : CAP_Config_Type := (ChannelA:=FALSE,ChannelB:=FALSE,ChannelC:=FALSE,HeadRotationDir:=FALSE,BufferSize:=0,PickAndPlace:=0,CamHeightPosition:=0);
	VAR_CAP_ActualConfig : CAP_Config_Type;
	VAR_Greasing_ModeInternal : INT;
	VAR_Greasing_ModeInternal2 : INT; (*//V4.A.A.1.6.11*)
	VAR_CAP_ModeActual : INT;
	VAR_SikoMultibody_ModeInternal : CAP_SikoMode_Type; (*V4.A.A.1.6.12*)
	VAR_CamSizeChange_ModeInternal : CAP_CamMode_Type;
	VAR_Buffer_ModeInternal : CAP_BufferMode_Type;
	VAR_Buffer_Empty : BOOL;
	VAR_Buffer_Lower : BOOL;
	VAR_CAP_GreasingWorkingSecond : UINT;
	VAR_CAP_GreasingWorkingHours : UINT;
	VAR_CAP_GreasingModeActual : UINT;
	VAR_CAP_GreasingModeActual2 : UINT; (*//V4.A.A.1.6.11*)
END_VAR
VAR
	CAP : CAP_Type;
	VAR_CAP_EquatoruqueCalModeSave : CAP_EquCalMode_Type; (*//V4.A.A.1.6.12*)
	VAR_CAP_EquatoruqueCalModeActual : CAP_EquCalMode_Type; (*//V4.A.A.1.6.12*)
	VAR_CAP_HeadData : ARRAY[0..48] OF CAP_Head_Type; (*//V4.A.A.1.6.12*)
END_VAR
VAR RETAIN
	VAR_CAP_Hopper_Running : BOOL; (*//v1.7.4 Tengo memoria di quale tramoggia sta lavorando 0=TramoggiaA  1=TramoggiaB*)
	VAR_HopperA_Empty : BOOL; (*//v1.7.4*)
	VAR_HopperB_Empty : BOOL; (*//v1.7.4*)
END_VAR
```

### CFG_Global.var
```iecst
VAR
	CFG_Par : CFG_Par_Type;
	CFG_ITC : CFG_ITC_Type;
	CFG_Cap_Par : CFG_Cap_Par_Type;
	CFG_Crw_Par : CFG_Crw_Par_Type;
	CFG_OPS : CFG_OPS_Type;
	CFG : CFG_Type;
END_VAR
```

### COP_Global.var
```iecst
VAR
	COP : COP_Type;
END_VAR
```

### CRW_Global.var
```iecst
VAR RETAIN
	VAR_CRW_ActualConfig : CRW_Config_Type;
	VAR_CRW_ModeActual : INT;
END_VAR
VAR
	CRW : CRW_Type;
END_VAR
```

### CSR_Global.var
```iecst
VAR RETAIN
	VAR_Lift_Sequencer : CSR_Lift_SeqMode_Type;
	VAR_CSR_Sequencer : CSR_Sequencer_Type;
END_VAR
VAR
	CSR : CSR_Type;
END_VAR
VAR RETAIN
	SIKO_AXIS2Data : SIKO_MASTER_Type; (*V4.A.A.1.6.12*)
	SIKO_AXIS1Data : SIKO_MASTER_Type; (*V4.A.A.1.6.12*)
END_VAR
```

### DMC_Global.var
```iecst
VAR RETAIN
	VAR_DMC_FmcComError : BOOL;
	VAR_DMC_SequenceStatus : DMC_Mode_Type;
	VAR_DMC_SequenceModeManual : DMC_ModeManualSequencerType;
	VAR_DMC_Sequence : DMC_SequencerType;
END_VAR
```

### FMC_Global.var
```iecst
VAR
	FMC : FMC_DataTo_Type;
	FmcFlr : FmcFlr_Type;
	FmcCommStatus : ITC_CommStatus_Type;
	FlrFmc : FlrFmc_Type;
END_VAR
(*Filling Valves Control*)
VAR
	FMC_FillingValves : ARRAY[1..200] OF FMC_ValvesControl_Type;
END_VAR
```

### GNS_Global.var
```iecst
VAR
	GNS : GNS_Type;
END_VAR
```

### ITC_Global.var
```iecst
VAR
	ITC : ITC_Type;
END_VAR
(*SKID COMMUNICATION*)
VAR
	SkdCommStatus : ITC_CommStatus_Type;
	SkdFlr : SidelPrcFlr_Type;
	FlrSkd : FlrSidelPrc_Type;
END_VAR
(*COREBLEND COMMUNICATION*)
VAR
	CrbCommStatus : ITC_CommStatus_Type;
	CrbFlr : SidelPrcFlr_Type;
	FlrCrb : FlrSidelPrc_Type;
END_VAR
(*CAPFEEDER COMMUNICATION*)
VAR
	CfdCommStatus : ITC_CommStatus_Type;
	CfdFlr : CfdFlr_Type;
	FlrCfd : FlrCfd_Type;
END_VAR
(*CAPFEEDER2 COMMUNICATION *)
VAR
	Cfd2CommStatus : ITC_CommStatus_Type; (*V4.A.A.1.7.0*)
	Cfd2Flr : CfdFlr_Type; (*V4.A.A.1.7.0*)
	FlrCfd2 : FlrCfd_Type; (*V4.A.A.1.7.0*)
END_VAR
(*CAPDIS COMMUNICATION V4.A.A.1.7.0*)
VAR
	CdsCommStatus : ITC_CommStatus_Type; (*V4.A.A.1.7.0*)
	CdsFlr : CdsFlr_Type; (*V4.A.A.1.7.0*)
	FlrCds : FlrCds_Type; (*V4.A.A.1.7.0*)
END_VAR
(*INLET CONVEYOR COMMUNICATION //V4.A.A.1.6.14*)
VAR
	CviCommStatus : ITC_CommStatus_Type;
	CviFlr : CviFlr_Type;
	FlrCvi : FlrCvi_Type;
END_VAR
(*OUTLET CONVEYOR COMMUNICATION*)
VAR
	CvoCommStatus : ITC_CommStatus_Type;
	CvoFlr : CvoFlr_Type;
	FlrCvo : FlrCvo_Type;
END_VAR
(*VACUUM BARRIER COMPANY*)
VAR
	VbcCommStatus : ITC_CommStatus_Type;
	VbcFlr : VbcFlr_Type;
	FlrVbc : FlrVbc_Type;
END_VAR
(*COP COMMUNICATION*)
VAR
	CopCommStatus : ITC_CommStatus_Type;
	CopFlr : CopFlr_Type;
	FlrCop : FlrCop_Type;
END_VAR
(*FULL CONTAINERS INSPECTOR*)
VAR
	FciCommStatus : ITC_CommStatus_Type;
	FciFlr : FciFlr_Type;
	FlrFci : FlrFci_Type;
END_VAR
(*PRODUCT CHANGE OVER*)
VAR
	IcoFlr : EIT_ChangeOver_From_Type;
	FlrIco : EIT_ChangeOver_To_Type;
END_VAR
(*UV LAMP CAPS TREATMENTS*)
VAR
	UvlCommStatus : ITC_CommStatus_Type;
	UvlFlr : UvlFlr_Type;
	FlrUvl : FlrUvl_Type;
END_VAR
(*CAP COMMUNICATION*)
VAR
	CapCommStatus : ITC_CommStatus_Type;
	CapFlr : CapFlr_Type;
	FlrCap : FlrCap_Type;
END_VAR
(*FLAVOR DOSER //V4.A.A.1.6.11*)
VAR
	DosCommStatus : ITC_CommStatus_Type;
	DosFlr : DosFlr_Type;
	FlrDos : FlrDos_Type;
END_VAR
(*DATA ACQUISITION //V4.A.A.1.6.14*)
VAR
	DaqCommStatus : ITC_CommStatus_Type;
	DaqFlr : DaqFlr_Type;
	FlrDaq : FlrDaq_Type;
END_VAR
(*SCC COMMUNICATION //V4.A.A.1.6.14*)
VAR
	FlrScc : ARRAY[0..100] OF UINT;
	FlrScc_AliveBit : BOOL;
	SccFlr : ARRAY[0..100] OF UINT;
	SccFlr_AliveBit : BOOL;
END_VAR
(*WTT COMMUNICATION*)
VAR
	WttCommStatus : ITC_CommStatus_Type; (*V4.A.A.1.7.0*)
	WttFlr : WttFlr_Type; (*V4.A.A.1.7.0*)
	FlrWtt : FlrWtt_Type; (*V4.A.A.1.7.0*)
END_VAR
(*CDR COMMUNICATION V4.A.A.1.7.0*)
VAR
	CdrCommStatus : ITC_CommStatus_Type;
	CdrFlr : CdrFlr_Type;
	FlrCdr : FlrCdr_Type;
END_VAR
(*PST COMMUNICATION*)
VAR
	PstCommStatus : ITC_CommStatus_Type; (*v999hema*)
	PstFlr : PstFlr_Type;
	FlrPst : FlrPst_Type;
END_VAR
```

### MAU_Global.var
```iecst
VAR
	VAR_SafeLogicStatus : SafeLogicStatus_Type;
	MAU_DumCon : MAU_DumCon_Type;
	MAU_LftCon : MAU_LftCon_Type;
	MAU_Ups : MAU_Ups_Type;
	MAU_Aux : MAU_Aux_Type; (*//1.7.2*)
	MAU_Tray : MAU_Tray_Type;
	MAU_Scheduler : MAU_Scheduler_Type; (*V1.7.4*)
END_VAR
```

### MC_Global.var
```iecst
VAR
	MC_InputOutput : ST_MotionInterface;
END_VAR
```

### MNM_Global.var
```iecst
VAR RETAIN
	VAR_MNM_CocleaPhasingByPassDone : BOOL;
	VAR_MNM_RinserPhasingByPassDone : BOOL;
	VAR_MNM_RinserPhasingHemaDone : BOOL;
	VAR_MNM_CocleaPhasingHemaDone : BOOL;
END_VAR
VAR
	MNM : MNM_Type;
END_VAR
VAR RETAIN
	VAR_MNM_RinserPhasingPerValue : REAL;
END_VAR
VAR
	VAR_MNM_AlarmTest : BOOL;
END_VAR
VAR RETAIN
	VAR_MNM_CocleaPhasingPerValue : REAL;
END_VAR
```

### MNT_Global.var
```iecst
VAR RETAIN
	VAR_MNT_Macao : HMI_Macao_Type;
END_VAR
VAR
	MNT : MNT_Type;
END_VAR
```

### OPS_Global.var
```iecst
VAR
	OPS : OPS_Type;
END_VAR
VAR RETAIN
	VAR_OPS_Permanent : INT; (*V4.A.A.1.6.12h*)
END_VAR
```

### RCP_Global.var
```iecst
VAR
	RCP : RCP_Type;
END_VAR
```

### RNS_Global.var
```iecst
VAR RETAIN
	VAR_RNS_SeqPermanent : SEQ_Permanent_Type;
END_VAR
VAR
	RNS : RNS_Type; (*V4.A.A.1.6.12*)
	VAR_RNS_RnsNozzleData : ARRAY[1..200] OF RNS_NozzleData_Type := [(Visibility:=TRUE,NozzleNumber:=1),(Visibility:=TRUE,NozzleNumber:=2),(Visibility:=TRUE,NozzleNumber:=3),(Visibility:=TRUE,NozzleNumber:=4),(Visibility:=TRUE,NozzleNumber:=5),(Visibility:=TRUE,NozzleNumber:=6),(Visibility:=TRUE,NozzleNumber:=7),(Visibility:=TRUE,NozzleNumber:=8),(Visibility:=TRUE,NozzleNumber:=9),(Visibility:=TRUE,NozzleNumber:=10),(Visibility:=TRUE,NozzleNumber:=11),(Visibility:=TRUE,NozzleNumber:=12),(Visibility:=TRUE,NozzleNumber:=13),(Visibility:=TRUE,NozzleNumber:=14),(Visibility:=TRUE,NozzleNumber:=15),(Visibility:=TRUE,NozzleNumber:=16),(Visibility:=TRUE,NozzleNumber:=17),(Visibility:=TRUE,NozzleNumber:=18),(Visibility:=TRUE,NozzleNumber:=19),(Visibility:=TRUE,NozzleNumber:=20),(Visibility:=TRUE,NozzleNumber:=21),(Visibility:=TRUE,NozzleNumber:=22),(Visibility:=TRUE,NozzleNumber:=23),(Visibility:=TRUE,NozzleNumber:=24),(Visibility:=TRUE,NozzleNumber:=25),(Visibility:=TRUE,NozzleNumber:=26),(Visibility:=TRUE,NozzleNumber:=27),(Visibility:=TRUE,NozzleNumber:=28),(Visibility:=TRUE,NozzleNumber:=29),(Visibility:=TRUE,NozzleNumber:=30),(Visibility:=TRUE,NozzleNumber:=31),(Visibility:=TRUE,NozzleNumber:=32),(Visibility:=TRUE,NozzleNumber:=33),(Visibility:=TRUE,NozzleNumber:=34),(Visibility:=TRUE,NozzleNumber:=35),(Visibility:=TRUE,NozzleNumber:=36),(Visibility:=TRUE,NozzleNumber:=37),(Visibility:=TRUE,NozzleNumber:=38),(Visibility:=TRUE,NozzleNumber:=39),(Visibility:=TRUE,NozzleNumber:=40),(Visibility:=TRUE,NozzleNumber:=41),(Visibility:=TRUE,NozzleNumber:=42),(Visibility:=TRUE,NozzleNumber:=43),(Visibility:=TRUE,NozzleNumber:=44),(Visibility:=TRUE,NozzleNumber:=45),(Visibility:=TRUE,NozzleNumber:=46),(Visibility:=TRUE,NozzleNumber:=47),(Visibility:=TRUE,NozzleNumber:=48),(Visibility:=TRUE,NozzleNumber:=49),(Visibility:=TRUE,NozzleNumber:=50),(Visibility:=TRUE,NozzleNumber:=51),(Visibility:=TRUE,NozzleNumber:=52),(Visibility:=TRUE,NozzleNumber:=53),(Visibility:=TRUE,NozzleNumber:=54),(Visibility:=TRUE,NozzleNumber:=55),(Visibility:=TRUE,NozzleNumber:=56),(Visibility:=TRUE,NozzleNumber:=57),(Visibility:=TRUE,NozzleNumber:=58),(Visibility:=TRUE,NozzleNumber:=59),(Visibility:=TRUE,NozzleNumber:=60),(Visibility:=TRUE,NozzleNumber:=61),(Visibility:=TRUE,NozzleNumber:=62),(Visibility:=TRUE,NozzleNumber:=63),(Visibility:=TRUE,NozzleNumber:=64),(Visibility:=TRUE,NozzleNumber:=65),(Visibility:=TRUE,NozzleNumber:=66),(Visibility:=TRUE,NozzleNumber:=67),(Visibility:=TRUE,NozzleNumber:=68),(Visibility:=TRUE,NozzleNumber:=69),(Visibility:=TRUE,NozzleNumber:=70),(Visibility:=TRUE,NozzleNumber:=71),(Visibility:=TRUE,NozzleNumber:=72),(Visibility:=TRUE,NozzleNumber:=73),(Visibility:=TRUE,NozzleNumber:=74),(Visibility:=TRUE,NozzleNumber:=75),(Visibility:=TRUE,NozzleNumber:=76),(Visibility:=TRUE,NozzleNumber:=77),(Visibility:=TRUE,NozzleNumber:=78),(Visibility:=TRUE,NozzleNumber:=79),(Visibility:=TRUE,NozzleNumber:=80),(Visibility:=TRUE,NozzleNumber:=81),(Visibility:=TRUE,NozzleNumber:=82),(Visibility:=TRUE,NozzleNumber:=83),(Visibility:=TRUE,NozzleNumber:=84),(Visibility:=TRUE,NozzleNumber:=85),(Visibility:=TRUE,NozzleNumber:=86),(Visibility:=TRUE,NozzleNumber:=87),(Visibility:=TRUE,NozzleNumber:=88),(Visibility:=TRUE,NozzleNumber:=89),(Visibility:=TRUE,NozzleNumber:=90),(Visibility:=TRUE,NozzleNumber:=91),(Visibility:=TRUE,NozzleNumber:=92),(Visibility:=TRUE,NozzleNumber:=93),(Visibility:=TRUE,NozzleNumber:=94),(Visibility:=TRUE,NozzleNumber:=95),(Visibility:=TRUE,NozzleNumber:=96),(Visibility:=TRUE,NozzleNumber:=97),(Visibility:=TRUE,NozzleNumber:=98),(Visibility:=TRUE,NozzleNumber:=99),(Visibility:=TRUE,NozzleNumber:=100),(Visibility:=TRUE,NozzleNumber:=101),(Visibility:=TRUE,NozzleNumber:=102),(Visibility:=TRUE,NozzleNumber:=103),(Visibility:=TRUE,NozzleNumber:=104),(Visibility:=TRUE,NozzleNumber:=105),(Visibility:=TRUE,NozzleNumber:=106),(Visibility:=TRUE,NozzleNumber:=107),(Visibility:=TRUE,NozzleNumber:=108),(Visibility:=TRUE,NozzleNumber:=109),(Visibility:=TRUE,NozzleNumber:=110),(Visibility:=TRUE,NozzleNumber:=111),(Visibility:=TRUE,NozzleNumber:=112),(Visibility:=TRUE,NozzleNumber:=113),(Visibility:=TRUE,NozzleNumber:=114),(Visibility:=TRUE,NozzleNumber:=115),(Visibility:=TRUE,NozzleNumber:=116),(Visibility:=TRUE,NozzleNumber:=117),(Visibility:=TRUE,NozzleNumber:=118),(Visibility:=TRUE,NozzleNumber:=119),(Visibility:=TRUE,NozzleNumber:=120),(Visibility:=FALSE,NozzleNumber:=121),79((0))]; (*V4.A.A.1.7.0*)
END_VAR
```

### SFT_Global.var
```iecst
VAR RETAIN
	VAR_SFT_FillerShift : ARRAY[1..CST_ShiftDimension] OF MachineShift_Type;
	VAR_SFT_ShiftStartPosition : INT;
	VAR_SFT_ShiftRinserControlAir : INT; (*V4.A.A.1.7.0*)
	VAR_SFT_ShiftRinserControlWater : INT; (*V4.A.A.1.7.0*)
	VAR_SFT_ShiftRinserControlIns : INT; (*V4.A.A.1.7.0*)
	VAR_SFT_NumberDmcInserted : INT;
	VAR_SFT_NumberDmcFirstHalIns : USINT;
	VAR_SFT_NumberDmcSecondHalIns : USINT;
END_VAR
(*FILLING VALVE DATA master nuovo*)
VAR RETAIN
	VAR_SFT_DummyIndexStartPos : INT;
	(*VAR_SFT_DummyContainerData : ARRAY[1..200] OF DummyContainerDataStructure_Type;*)
	VAR_SFT_FillingValveData : ARRAY[1..150] OF FillingValveDataStructure_Type;
END_VAR
VAR
	SFT : SFT_Type;
END_VAR
```

### TNK_Global.var
```iecst
VAR
	TNK : TNK_Type;
END_VAR
```

### DOS_Global.var
```iecst
VAR RETAIN
	VAR_DOS_SeqPermanent : SEQ_Permanent_Type; (*v999hema*)
	VAR_DOS_CamPermanent : SEQ_Permanent_Type;
	VAR_DOS_MotPermanent : SEQ_Permanent_Type;
END_VAR
VAR
	DOS : DOS_Type;
END_VAR
VAR RETAIN
	Delta_205MEF : REAL;
	Delta_206MEF : REAL;
END_VAR
```

### REL_Global.var
```iecst
VAR
	REL : REL_Type;
END_VAR
```

### BTC_Global.var - not listed in the package file held
```iecst
VAR RETAIN
	VAR_BTC_SeqPermanent : SEQ_Permanent_Type;
END_VAR
VAR
	BTC : BTC_Type;
END_VAR
```

### EIT_Global.var - not listed in the package file held
```iecst
(*OPC VARIABLES - CHANGE THEM REQUIRES TO CHANGE OPC CONFIGURATION AND A WARM RESTART*)
VAR
	VAR_EIT : EIT_Type;
	VAR_ChangeOver : EIT_ChangeOver_Type;
	VAR_PackMLv30 : EIT_OMAC_Type;
	VAR_WS : WS_Type;
END_VAR
(*PowerMeter IO Var*)
VAR
	VAR_ECO_RDirectRead : ARRAY[0..4] OF REAL;
	VAR_ECO_IDirectRead : ARRAY[0..4] OF UDINT;
END_VAR
```

### ICO_Global.var - not listed in the package file held
```iecst
VAR
	ICO : ICO_Type;
END_VAR
```

### Package Logical/00_AID/Libraries/Sidel_Libraries - Sidel libraries

### Library Logical/00_AID/Libraries/Sidel_Libraries/Powertoys (IEC, version 1.05.0) - Set of tools
Depends on: AsIODiag, AsArProf, AsARCfg, AsArSdm, FileIO

#### Powertoys.typ - Exported data types
```iecst
(********************************************************************
 * COPYRIGHT -- Bernecker + Rainer
 ********************************************************************
 * Library: Powertoys
 * File: Powertoys.typ
 * Author: gibertinim
 * Created: March 27, 2014
 ********************************************************************
 * Data types of library Powertoys
 ********************************************************************)
(********************************                    CUSTOM LOGGER ENTRY                   ***********************************************************)

TYPE
	pwr_log_custom_entry : 	STRUCT  (*Custom logger entry string*)
		adr_string : UDINT; (*Address of the ascii string*)
		len : UDINT; (*Length of the binary memory data*)
		adr_mem : UDINT; (*Address to the binary memory data*)
		errorNum : UINT; (*Error number to write*)
		logLevel : USINT; (*Information level*)
	END_STRUCT;
END_TYPE

(*********************************                            HARDWARE LIST                          **************************************************************)

TYPE
	searchIO_info_typ : 	STRUCT  (*Hardware information list*)
		Path : STRING[80]; (*Station path*)
		ModelNumber : STRING[80]; (*Model number*)
		Name : STRING[80]; (*Hw name*)
		Serial : UDINT; (*Serial number*)
	END_STRUCT;
END_TYPE

(********************************                              AXIS INFORMATIONS                **************************************************************)

TYPE
	pwlInfo_typ : 	STRUCT  (*Powerlink node properties datatype*)
		number : USINT; (*Number of Powerlink Module*)
		path : STRING[80]; (*Path of Powerlink Module*)
		description : STRING[80]; (*Description of Powerlink Module*)
		name : STRING[80]; (*Name of Powerlink Module*)
		modelNumber : STRING[80]; (*Module number of powerlink *)
		present : BOOL; (*Enable blinking*)
	END_STRUCT;
END_TYPE
```

#### Powertoys.var - Exported constants
```iecst
(********************************************************************
 * COPYRIGHT -- Bernecker + Rainer
 ********************************************************************
 * Library: Powertoys
 * File: Powertoys.var
 * Author: gibertinim
 * Created: March 27, 2014
 ********************************************************************
 * Constants of library Powertoys
 ********************************************************************)
VAR CONSTANT
	CST_SW_OBJ_CHANGED : UINT := 55100; (*Software object changed*)
	CST_SDM_DISABLE : UINT := 55110; (*Disable SDM*)
	CST_SDM_ACTIVE : UINT := 55111; (*Activate SDM*)
	CST_SDM_DUMP_DONE : UINT := 55112; (*System dump completed*)
	CST_NO_NTC : UINT := 55120; (*No network command trace available*)
END_VAR
```
